LIN {X 0,Y 228.257,Z 260.465,A -85,B 0,C 180,E1 -20025.086,E2 -20025.086} C_VEL
LIN {X 0,Y 228.489,Z 263.113,A -85,B 0,C 180,E1 -20029.335,E2 -20029.335} C_VEL
LIN {X 0,Y 229.645,Z 266.297,A -85,B 0,C 180,E1 -20029.751,E2 -20029.751} C_VEL
LIN {X 0,Y 231.014,Z 268.634,A -85,B 0,C 180,E1 -20030.164,E2 -20030.164} C_VEL
LIN {X 0,Y 235.943,Z 279.475,A -85,B 0,C 180,E1 -20031.89,E2 -20031.89} C_VEL
LIN {X 0,Y 239.913,Z 290.987,A -85,B 0,C 180,E1 -20033.668,E2 -20033.668} C_VEL
LIN {X 0,Y 242.925,Z 302.472,A -85,B 0,C 180,E1 -20035.491,E2 -20035.491} C_VEL
LIN {X 0,Y 244.896,Z 313.256,A -85,B 0,C 180,E1 -20037.287,E2 -20037.287} C_VEL
LIN {X 0,Y 245.991,Z 323.127,A -85,B 0,C 180,E1 -20039.052,E2 -20039.052} C_VEL
LIN {X 0,Y 245.201,Z 327.647,A -85,B 0,C 180,E1 -20039.767,E2 -20039.767} C_VEL
LIN {X 0,Y 242.212,Z 338.615,A -85,B 0,C 180,E1 -20041.632,E2 -20041.632} C_VEL
LIN {X 0,Y 239.048,Z 349.08,A -85,B 0,C 180,E1 -20043.832,E2 -20043.832} C_VEL
LIN {X 0,Y 235.989,Z 358.524,A -85,B 0,C 180,E1 -20046.294,E2 -20046.294} C_VEL
LIN {X 0,Y 233.317,Z 366.346,A -85,B 0,C 180,E1 -20048.81,E2 -20048.81} C_VEL
LIN {X 0,Y 231.34,Z 372.844,A -85,B 0,C 180,E1 -20051.399,E2 -20051.399} C_VEL
LIN {X 0,Y 229.395,Z 378.242,A -85,B 0,C 180,E1 -20053.994,E2 -20053.994} C_VEL
LIN {X 0,Y 227.608,Z 383.911,A -85,B 0,C 180,E1 -20057.518,E2 -20057.518} C_VEL
LIN {X 0,Y 226.471,Z 388.027,A -85,B 0,C 180,E1 -20061.074,E2 -20061.074} C_VEL
LIN {X 0,Y 225.835,Z 390.798,A -85,B 0,C 180,E1 -20064.777,E2 -20064.777} C_VEL
LIN {X 0,Y 225.647,Z 392.058,A -85,B 0,C 180,E1 -20068.215,E2 -20068.215} C_VEL
LIN {X 0,Y 225.667,Z 392.235,A -85,B 0,C 180,E1 -20070,E2 -20070} C_VEL
LIN {X 0,Y 225.703,Z 391.606,A -85,B 0,C 180,E1 -20073.571,E2 -20073.571} C_VEL
LIN {X 0,Y 226.103,Z 389.645,A -85,B 0,C 180,E1 -20077.142,E2 -20077.142} C_VEL
LIN {X 0,Y 226.949,Z 386.307,A -85,B 0,C 180,E1 -20080.708,E2 -20080.708} C_VEL
LIN {X 0,Y 228.318,Z 381.491,A -85,B 0,C 180,E1 -20084.256,E2 -20084.256} C_VEL
LIN {X 0,Y 230.642,Z 375.034,A -85,B 0,C 180,E1 -20087.741,E2 -20087.741} C_VEL
LIN {X 0,Y 232.661,Z 368.29,A -85,B 0,C 180,E1 -20090.606,E2 -20090.606} C_VEL
LIN {X 0,Y 235.407,Z 360.312,A -85,B 0,C 180,E1 -20093.302,E2 -20093.302} C_VEL
LIN {X 0,Y 238.452,Z 351.255,A -85,B 0,C 180,E1 -20095.769,E2 -20095.769} C_VEL
LIN {X 0,Y 241.791,Z 340.283,A -85,B 0,C 180,E1 -20098.186,E2 -20098.186} C_VEL
LIN {X 0,Y 244.745,Z 329.799,A -85,B 0,C 180,E1 -20100.029,E2 -20100.029} C_VEL
LIN {X 0,Y 246.084,Z 323.924,A -85,B 0,C 180,E1 -20100.936,E2 -20100.936} C_VEL
LIN {X 0,Y 245.035,Z 313.632,A -85,B 0,C 180,E1 -20102.773,E2 -20102.773} C_VEL
LIN {X 0,Y 242.991,Z 302.457,A -85,B 0,C 180,E1 -20104.644,E2 -20104.644} C_VEL
LIN {X 0,Y 239.709,Z 289.968,A -85,B 0,C 180,E1 -20106.619,E2 -20106.619} C_VEL
LIN {X 0,Y 235.279,Z 277.883,A -85,B 0,C 180,E1 -20108.509,E2 -20108.509} C_VEL
LIN {X 0,Y 232.127,Z 271.034,A -85,B 0,C 180,E1 -20109.612,E2 -20109.612} C_VEL
LIN {X 0,Y 230.198,Z 267.155,A -85,B 0,C 180,E1 -20110.247,E2 -20110.247} C_VEL
LIN {X 0,Y 228.812,Z 264.447,A -85,B 0,C 180,E1 -20110.674,E2 -20110.674} C_VEL
LIN {X 0,Y 228.503,Z 263.113,A -85,B 0,C 180,E1 -20110.832,E2 -20110.832} C_VEL
LIN {X 0,Y 228.241,Z 260.465,A -85,B 0,C 180,E1 -20115.09,E2 -20115.09} C_VEL
LIN {X 0,Y 227.843,Z 257.899,A -85,B 0,C 180,E1 -20119.627,E2 -20119.627} C_VEL
LIN {X 0,Y 227.867,Z 257.727,A -85,B 0,C 180,E1 -20124.125,E2 -20124.125} C_VEL
LIN {X 0,Y 227.873,Z 257.726,A -85,B 0,C 180,E1 -20128.378,E2 -20128.378} C_VEL
LIN {X 0,Y 227.888,Z 257.724,A -85,B 0,C 180,E1 -20132.445,E2 -20132.445} C_VEL
LIN {X 0,Y 227.909,Z 257.721,A -85,B 0,C 180,E1 -20136.367,E2 -20136.367} C_VEL
LIN {X 0,Y 227.941,Z 257.715,A -85,B 0,C 180,E1 -20140.174,E2 -20140.174} C_VEL
LIN {X 0,Y 228.061,Z 257.701,A -85,B 0,C 180,E1 -20143.898,E2 -20143.898} C_VEL
LIN {X 0,Y 228.075,Z 257.701,A -85,B 0,C 180,E1 -20147.543,E2 -20147.543} C_VEL
LIN {X 0,Y 228.266,Z 257.676,A -85,B 0,C 180,E1 -20151.144,E2 -20151.144} C_VEL
LIN {X 0,Y 228.321,Z 257.67,A -85,B 0,C 180,E1 -20152.927,E2 -20152.927} C_VEL
LIN {X 0,Y 228.552,Z 257.641,A -85,B 0,C 180,E1 -20158.238,E2 -20158.238} C_VEL
LIN {X 0,Y 228.555,Z 257.64,A -85,B 0,C 180,E1 -20161.762,E2 -20161.762} C_VEL
LIN {X 0,Y 228.31,Z 257.669,A -85,B 0,C 180,E1 -20167.073,E2 -20167.073} C_VEL
LIN {X 0,Y 228.145,Z 257.692,A -85,B 0,C 180,E1 -20170.651,E2 -20170.651} C_VEL
LIN {X 0,Y 228.041,Z 257.705,A -85,B 0,C 180,E1 -20174.273,E2 -20174.273} C_VEL
LIN {X 0,Y 227.97,Z 257.715,A -85,B 0,C 180,E1 -20177.956,E2 -20177.956} C_VEL
LIN {X 0,Y 227.922,Z 257.72,A -85,B 0,C 180,E1 -20182.323,E2 -20182.323} C_VEL
LIN {X 0,Y 227.924,Z 257.714,A -85,B 0,C 180,E1 -20186.592,E2 -20186.592} C_VEL
LIN {X 0,Y 227.875,Z 257.726,A -85,B 0,C 180,E1 -20190.28,E2 -20190.28} C_VEL
LIN {X 0,Y 227.857,Z 257.724,A -85,B 0,C 180,E1 -20191.624,E2 -20191.624} C_VEL
LIN {X 0,Y 227.976,Z 258.28,A -85,B 0,C 180,E1 -20193.704,E2 -20193.704} C_VEL
LIN {X 0,Y 228.398,Z 260.942,A -85,B 0,C 180,E1 -20197.982,E2 -20197.982} C_VEL
LIN {X 0,Y 228.903,Z 264.055,A -85,B 0,C 180,E1 -20202.534,E2 -20202.534} C_VEL
LIN {X 0,Y 229.191,Z 265.956,A -85,B 0,C 180,E1 -20205.147,E2 -20205.147} C_VEL
LIN {X 0,Y 229.35,Z 268.73,A -85,B 0,C 180,E1 -20208.665,E2 -20208.665} C_VEL
LIN {X 0,Y 229.788,Z 269.831,A -85,B 0,C 180,E1 -20209.268,E2 -20209.268} C_VEL
LIN {X 0,Y 230.97,Z 272.393,A -85,B 0,C 180,E1 -20209.868,E2 -20209.868} C_VEL
LIN {X 0,Y 232.259,Z 276.618,A -85,B 0,C 180,E1 -20210.386,E2 -20210.386} C_VEL
LIN {X 0,Y 232.855,Z 282.514,A -85,B 0,C 180,E1 -20210.851,E2 -20210.851} C_VEL
LIN {X 0,Y 232.552,Z 288.953,A -85,B 0,C 180,E1 -20211.289,E2 -20211.289} C_VEL
LIN {X 0,Y 232.587,Z 295.048,A -85,B 0,C 180,E1 -20211.896,E2 -20211.896} C_VEL
LIN {X 0,Y 232.958,Z 296.91,A -85,B 0,C 180,E1 -20212.162,E2 -20212.162} C_VEL
LIN {X 0,Y 235.613,Z 308.607,A -85,B 0,C 180,E1 -20213.985,E2 -20213.985} C_VEL
LIN {X 0,Y 237.168,Z 319.32,A -85,B 0,C 180,E1 -20215.734,E2 -20215.734} C_VEL
LIN {X 0,Y 238.014,Z 331.504,A -85,B 0,C 180,E1 -20217.893,E2 -20217.893} C_VEL
LIN {X 0,Y 237.956,Z 336.523,A -85,B 0,C 180,E1 -20218.839,E2 -20218.839} C_VEL
LIN {X 0,Y 234.74,Z 348.029,A -85,B 0,C 180,E1 -20220.888,E2 -20220.888} C_VEL
LIN {X 0,Y 231.105,Z 359.097,A -85,B 0,C 180,E1 -20223.349,E2 -20223.349} C_VEL
LIN {X 0,Y 228.033,Z 368.236,A -85,B 0,C 180,E1 -20225.897,E2 -20225.897} C_VEL
LIN {X 0,Y 225.047,Z 376.976,A -85,B 0,C 180,E1 -20228.953,E2 -20228.953} C_VEL
LIN {X 0,Y 223.05,Z 383.133,A -85,B 0,C 180,E1 -20231.634,E2 -20231.634} C_VEL
LIN {X 0,Y 220.835,Z 389.674,A -85,B 0,C 180,E1 -20235.25,E2 -20235.25} C_VEL
LIN {X 0,Y 219.427,Z 394.573,A -85,B 0,C 180,E1 -20238.92,E2 -20238.92} C_VEL
LIN {X 0,Y 218.684,Z 397.982,A -85,B 0,C 180,E1 -20242.614,E2 -20242.614} C_VEL
LIN {X 0,Y 218.48,Z 399.737,A -85,B 0,C 180,E1 -20245.71,E2 -20245.71} C_VEL
LIN {X 0,Y 218.469,Z 400.5,A -85,B 0,C 180,E1 -20248.156,E2 -20248.156} C_VEL
LIN {X 0,Y 218.574,Z 400.666,A -85,B 0,C 180,E1 -20250,E2 -20250} C_VEL
LIN {X 0,Y 218.449,Z 399.983,A -85,B 0,C 180,E1 -20253.689,E2 -20253.689} C_VEL
LIN {X 0,Y 218.684,Z 397.952,A -85,B 0,C 180,E1 -20257.386,E2 -20257.386} C_VEL
LIN {X 0,Y 219.415,Z 394.525,A -85,B 0,C 180,E1 -20261.08,E2 -20261.08} C_VEL
LIN {X 0,Y 220.828,Z 389.603,A -85,B 0,C 180,E1 -20264.75,E2 -20264.75} C_VEL
LIN {X 0,Y 223.041,Z 383.044,A -85,B 0,C 180,E1 -20268.367,E2 -20268.367} C_VEL
LIN {X 0,Y 225.382,Z 375.745,A -85,B 0,C 180,E1 -20271.493,E2 -20271.493} C_VEL
LIN {X 0,Y 228.498,Z 366.709,A -85,B 0,C 180,E1 -20274.533,E2 -20274.533} C_VEL
LIN {X 0,Y 231.657,Z 357.234,A -85,B 0,C 180,E1 -20277.069,E2 -20277.069} C_VEL
LIN {X 0,Y 235.087,Z 346.749,A -85,B 0,C 180,E1 -20279.31,E2 -20279.31} C_VEL
LIN {X 0,Y 237.729,Z 337.361,A -85,B 0,C 180,E1 -20280.982,E2 -20280.982} C_VEL
LIN {X 0,Y 237.869,Z 329.442,A -85,B 0,C 180,E1 -20282.438,E2 -20282.438} C_VEL
LIN {X 0,Y 236.904,Z 317.539,A -85,B 0,C 180,E1 -20284.513,E2 -20284.513} C_VEL
LIN {X 0,Y 235.241,Z 306.98,A -85,B 0,C 180,E1 -20286.231,E2 -20286.231} C_VEL
LIN {X 0,Y 232.694,Z 296.172,A -85,B 0,C 180,E1 -20287.903,E2 -20287.903} C_VEL
LIN {X 0,Y 229.123,Z 285.061,A -85,B 0,C 180,E1 -20289.607,E2 -20289.607} C_VEL
LIN {X 0,Y 225.78,Z 277.127,A -85,B 0,C 180,E1 -20290.878,E2 -20290.878} C_VEL
LIN {X 0,Y 224.135,Z 273.5,A -85,B 0,C 180,E1 -20291.464,E2 -20291.464} C_VEL
LIN {X 0,Y 222.625,Z 270.595,A -85,B 0,C 180,E1 -20291.953,E2 -20291.953} C_VEL
LIN {X 0,Y 222.315,Z 269.109,A -85,B 0,C 180,E1 -20292.166,E2 -20292.166} C_VEL
LIN {X 0,Y 221.999,Z 266.349,A -85,B 0,C 180,E1 -20295.855,E2 -20295.855} C_VEL
LIN {X 0,Y 221.579,Z 263.09,A -85,B 0,C 180,E1 -20300.628,E2 -20300.628} C_VEL
LIN {X 0,Y 221.102,Z 260.321,A -85,B 0,C 180,E1 -20305.1,E2 -20305.1} C_VEL
LIN {X 0,Y 220.88,Z 259.101,A -85,B 0,C 180,E1 -20307.255,E2 -20307.255} C_VEL
LIN {X 0,Y 220.834,Z 258.604,A -85,B 0,C 180,E1 -20309.39,E2 -20309.39} C_VEL
LIN {X 0,Y 220.876,Z 258.597,A -85,B 0,C 180,E1 -20313.547,E2 -20313.547} C_VEL
LIN {X 0,Y 220.867,Z 258.599,A -85,B 0,C 180,E1 -20317.552,E2 -20317.552} C_VEL
LIN {X 0,Y 220.931,Z 258.586,A -85,B 0,C 180,E1 -20322.617,E2 -20322.617} C_VEL
LIN {X 0,Y 221.004,Z 258.581,A -85,B 0,C 180,E1 -20327.138,E2 -20327.138} C_VEL
LIN {X 0,Y 221.198,Z 258.556,A -85,B 0,C 180,E1 -20330.859,E2 -20330.859} C_VEL
LIN {X 0,Y 221.127,Z 258.565,A -85,B 0,C 180,E1 -20334.529,E2 -20334.529} C_VEL
LIN {X 0,Y 221.511,Z 258.519,A -85,B 0,C 180,E1 -20338.182,E2 -20338.182} C_VEL
LIN {X 0,Y 221.511,Z 258.516,A -85,B 0,C 180,E1 -20341.818,E2 -20341.818} C_VEL
LIN {X 0,Y 221.261,Z 258.549,A -85,B 0,C 180,E1 -20347.3,E2 -20347.3} C_VEL
LIN {X 0,Y 221.083,Z 258.571,A -85,B 0,C 180,E1 -20350.996,E2 -20350.996} C_VEL
LIN {X 0,Y 221.018,Z 258.58,A -85,B 0,C 180,E1 -20356.63,E2 -20356.63} C_VEL
LIN {X 0,Y 220.886,Z 258.594,A -85,B 0,C 180,E1 -20360.487,E2 -20360.487} C_VEL
LIN {X 0,Y 220.864,Z 258.597,A -85,B 0,C 180,E1 -20364.436,E2 -20364.436} C_VEL
LIN {X 0,Y 220.828,Z 258.603,A -85,B 0,C 180,E1 -20368.515,E2 -20368.515} C_VEL
LIN {X 0,Y 220.817,Z 258.604,A -85,B 0,C 180,E1 -20372.756,E2 -20372.756} C_VEL
LIN {X 0,Y 220.802,Z 258.607,A -85,B 0,C 180,E1 -20377.275,E2 -20377.275} C_VEL
LIN {X 0,Y 220.796,Z 258.683,A -85,B 0,C 180,E1 -20379.539,E2 -20379.539} C_VEL
LIN {X 0,Y 221.19,Z 261.272,A -85,B 0,C 180,E1 -20384.349,E2 -20384.349} C_VEL
LIN {X 0,Y 221.465,Z 263.28,A -85,B 0,C 180,E1 -20387.742,E2 -20387.742} C_VEL
LIN {X 0,Y 222.597,Z 266.399,A -85,B 0,C 180,E1 -20388.192,E2 -20388.192} C_VEL
LIN {X 0,Y 224.096,Z 268.756,A -85,B 0,C 180,E1 -20388.667,E2 -20388.667} C_VEL
LIN {X 0,Y 229.315,Z 279.77,A -85,B 0,C 180,E1 -20390.589,E2 -20390.589} C_VEL
LIN {X 0,Y 233.519,Z 291.493,A -85,B 0,C 180,E1 -20392.542,E2 -20392.542} C_VEL
LIN {X 0,Y 236.826,Z 304.525,A -85,B 0,C 180,E1 -20394.721,E2 -20394.721} C_VEL
LIN {X 0,Y 238.737,Z 315.837,A -85,B 0,C 180,E1 -20396.724,E2 -20396.724} C_VEL
LIN {X 0,Y 239.585,Z 325.305,A -85,B 0,C 180,E1 -20398.507,E2 -20398.507} C_VEL
LIN {X 0,Y 236.916,Z 335.554,A -85,B 0,C 180,E1 -20400.206,E2 -20400.206} C_VEL
LIN {X 0,Y 233.85,Z 345.666,A -85,B 0,C 180,E1 -20402.236,E2 -20402.236} C_VEL
LIN {X 0,Y 230.562,Z 355.7,A -85,B 0,C 180,E1 -20404.739,E2 -20404.739} C_VEL
LIN {X 0,Y 227.557,Z 364.031,A -85,B 0,C 180,E1 -20407.291,E2 -20407.291} C_VEL
LIN {X 0,Y 224.829,Z 371.981,A -85,B 0,C 180,E1 -20410.364,E2 -20410.364} C_VEL
LIN {X 0,Y 223.217,Z 376.707,A -85,B 0,C 180,E1 -20412.596,E2 -20412.596} C_VEL
LIN {X 0,Y 221.447,Z 381.418,A -85,B 0,C 180,E1 -20415.292,E2 -20415.292} C_VEL
LIN {X 0,Y 219.965,Z 386.291,A -85,B 0,C 180,E1 -20418.948,E2 -20418.948} C_VEL
LIN {X 0,Y 219.049,Z 389.679,A -85,B 0,C 180,E1 -20422.627,E2 -20422.627} C_VEL
LIN {X 0,Y 218.622,Z 391.687,A -85,B 0,C 180,E1 -20426.314,E2 -20426.314} C_VEL
LIN {X 0,Y 218.585,Z 392.369,A -85,B 0,C 180,E1 -20430,E2 -20430} C_VEL
LIN {X 0,Y 218.62,Z 391.74,A -85,B 0,C 180,E1 -20433.687,E2 -20433.687} C_VEL
LIN {X 0,Y 219.049,Z 389.78,A -85,B 0,C 180,E1 -20437.374,E2 -20437.374} C_VEL
LIN {X 0,Y 219.951,Z 386.442,A -85,B 0,C 180,E1 -20441.053,E2 -20441.053} C_VEL
LIN {X 0,Y 221.41,Z 381.625,A -85,B 0,C 180,E1 -20444.711,E2 -20444.711} C_VEL
LIN {X 0,Y 223.874,Z 375.168,A -85,B 0,C 180,E1 -20448.296,E2 -20448.296} C_VEL
LIN {X 0,Y 225.91,Z 368.651,A -85,B 0,C 180,E1 -20451.154,E2 -20451.154} C_VEL
LIN {X 0,Y 228.901,Z 360.444,A -85,B 0,C 180,E1 -20454.005,E2 -20454.005} C_VEL
LIN {X 0,Y 232.053,Z 351.388,A -85,B 0,C 180,E1 -20456.534,E2 -20456.534} C_VEL
LIN {X 0,Y 235.555,Z 340.414,A -85,B 0,C 180,E1 -20459.002,E2 -20459.002} C_VEL
LIN {X 0,Y 238.814,Z 329.133,A -85,B 0,C 180,E1 -20461.014,E2 -20461.014} C_VEL
LIN {X 0,Y 239.666,Z 324.668,A -85,B 0,C 180,E1 -20461.744,E2 -20461.744} C_VEL
LIN {X 0,Y 238.534,Z 313.568,A -85,B 0,C 180,E1 -20463.818,E2 -20463.818} C_VEL
LIN {X 0,Y 236.426,Z 302.352,A -85,B 0,C 180,E1 -20465.784,E2 -20465.784} C_VEL
LIN {X 0,Y 233.712,Z 292.001,A -85,B 0,C 180,E1 -20467.52,E2 -20467.52} C_VEL
LIN {X 0,Y 229.307,Z 279.636,A -85,B 0,C 180,E1 -20469.58,E2 -20469.58} C_VEL
LIN {X 0,Y 225.292,Z 271.3,A -85,B 0,C 180,E1 -20471.058,E2 -20471.058} C_VEL
LIN {X 0,Y 223.483,Z 267.64,A -85,B 0,C 180,E1 -20471.703,E2 -20471.703} C_VEL
LIN {X 0,Y 221.854,Z 264.855,A -85,B 0,C 180,E1 -20472.224,E2 -20472.224} C_VEL
LIN {X 0,Y 221.446,Z 263.285,A -85,B 0,C 180,E1 -20472.425,E2 -20472.425} C_VEL
LIN {X 0,Y 221.076,Z 260.645,A -85,B 0,C 180,E1 -20476.985,E2 -20476.985} C_VEL
LIN {X 0,Y 220.812,Z 258.778,A -85,B 0,C 180,E1 -20480.464,E2 -20480.464} C_VEL
LIN {X 0,Y 220.826,Z 258.604,A -85,B 0,C 180,E1 -20482.793,E2 -20482.793} C_VEL
LIN {X 0,Y 220.82,Z 258.605,A -85,B 0,C 180,E1 -20487.244,E2 -20487.244} C_VEL
LIN {X 0,Y 220.839,Z 258.602,A -85,B 0,C 180,E1 -20491.487,E2 -20491.487} C_VEL
LIN {X 0,Y 220.865,Z 258.593,A -85,B 0,C 180,E1 -20495.565,E2 -20495.565} C_VEL
LIN {X 0,Y 220.888,Z 258.594,A -85,B 0,C 180,E1 -20499.513,E2 -20499.513} C_VEL
LIN {X 0,Y 221.019,Z 258.58,A -85,B 0,C 180,E1 -20503.37,E2 -20503.37} C_VEL
LIN {X 0,Y 221.014,Z 258.578,A -85,B 0,C 180,E1 -20507.139,E2 -20507.139} C_VEL
LIN {X 0,Y 221.204,Z 258.556,A -85,B 0,C 180,E1 -20510.859,E2 -20510.859} C_VEL
LIN {X 0,Y 221.257,Z 258.549,A -85,B 0,C 180,E1 -20512.7,E2 -20512.7} C_VEL
LIN {X 0,Y 221.51,Z 258.518,A -85,B 0,C 180,E1 -20518.182,E2 -20518.182} C_VEL
LIN {X 0,Y 221.513,Z 258.517,A -85,B 0,C 180,E1 -20521.818,E2 -20521.818} C_VEL
LIN {X 0,Y 221.247,Z 258.549,A -85,B 0,C 180,E1 -20527.3,E2 -20527.3} C_VEL
LIN {X 0,Y 221.065,Z 258.575,A -85,B 0,C 180,E1 -20530.996,E2 -20530.996} C_VEL
LIN {X 0,Y 220.988,Z 258.582,A -85,B 0,C 180,E1 -20536.632,E2 -20536.632} C_VEL
LIN {X 0,Y 220.882,Z 258.596,A -85,B 0,C 180,E1 -20540.487,E2 -20540.487} C_VEL
LIN {X 0,Y 220.849,Z 258.598,A -85,B 0,C 180,E1 -20544.437,E2 -20544.437} C_VEL
LIN {X 0,Y 220.806,Z 258.605,A -85,B 0,C 180,E1 -20548.518,E2 -20548.518} C_VEL
LIN {X 0,Y 220.82,Z 258.602,A -85,B 0,C 180,E1 -20550.758,E2 -20550.758} C_VEL
LIN {X 0,Y 220.894,Z 259.155,A -85,B 0,C 180,E1 -20552.743,E2 -20552.743} C_VEL
LIN {X 0,Y 221.399,Z 261.939,A -85,B 0,C 180,E1 -20557.477,E2 -20557.477} C_VEL
LIN {X 0,Y 221.797,Z 264.734,A -85,B 0,C 180,E1 -20561.714,E2 -20561.714} C_VEL
LIN {X 0,Y 222.221,Z 267.707,A -85,B 0,C 180,E1 -20565.911,E2 -20565.911} C_VEL
LIN {X 0,Y 222.335,Z 269.174,A -85,B 0,C 180,E1 -20567.836,E2 -20567.836} C_VEL
LIN {X 0,Y 223.344,Z 272.251,A -85,B 0,C 180,E1 -20568.223,E2 -20568.223} C_VEL
LIN {X 0,Y 224.813,Z 274.705,A -85,B 0,C 180,E1 -20568.683,E2 -20568.683} C_VEL
LIN {X 0,Y 229.334,Z 285.417,A -85,B 0,C 180,E1 -20570.399,E2 -20570.399} C_VEL
LIN {X 0,Y 232.958,Z 296.91,A -85,B 0,C 180,E1 -20572.162,E2 -20572.162} C_VEL
LIN {X 0,Y 233.805,Z 302.011,A -85,B 0,C 180,E1 -20572.867,E2 -20572.867} C_VEL
LIN {X 0,Y 233.669,Z 307.392,A -85,B 0,C 180,E1 -20573.483,E2 -20573.483} C_VEL
LIN {X 0,Y 231.828,Z 318.322,A -85,B 0,C 180,E1 -20574.699,E2 -20574.699} C_VEL
LIN {X 0,Y 231.236,Z 323.452,A -85,B 0,C 180,E1 -20575.428,E2 -20575.428} C_VEL
LIN {X 0,Y 231.257,Z 325.088,A -85,B 0,C 180,E1 -20575.704,E2 -20575.704} C_VEL
LIN {X 0,Y 231.615,Z 336.926,A -85,B 0,C 180,E1 -20577.992,E2 -20577.992} C_VEL
LIN {X 0,Y 228.544,Z 347.897,A -85,B 0,C 180,E1 -20580.019,E2 -20580.019} C_VEL
LIN {X 0,Y 224.74,Z 358.964,A -85,B 0,C 180,E1 -20582.531,E2 -20582.531} C_VEL
LIN {X 0,Y 221.544,Z 368.103,A -85,B 0,C 180,E1 -20585.144,E2 -20585.144} C_VEL
LIN {X 0,Y 218.375,Z 376.841,A -85,B 0,C 180,E1 -20588.278,E2 -20588.278} C_VEL
LIN {X 0,Y 216.272,Z 382.999,A -85,B 0,C 180,E1 -20591.037,E2 -20591.037} C_VEL
LIN {X 0,Y 213.926,Z 389.539,A -85,B 0,C 180,E1 -20594.762,E2 -20594.762} C_VEL
LIN {X 0,Y 212.413,Z 394.438,A -85,B 0,C 180,E1 -20598.549,E2 -20598.549} C_VEL
LIN {X 0,Y 211.624,Z 397.848,A -85,B 0,C 180,E1 -20602.366,E2 -20602.366} C_VEL
LIN {X 0,Y 211.387,Z 399.734,A -85,B 0,C 180,E1 -20605.876,E2 -20605.876} C_VEL
LIN {X 0,Y 211.373,Z 400.366,A -85,B 0,C 180,E1 -20608.094,E2 -20608.094} C_VEL
LIN {X 0,Y 211.473,Z 400.531,A -85,B 0,C 180,E1 -20610,E2 -20610} C_VEL
LIN {X 0,Y 211.355,Z 399.848,A -85,B 0,C 180,E1 -20613.813,E2 -20613.813} C_VEL
LIN {X 0,Y 211.623,Z 397.816,A -85,B 0,C 180,E1 -20617.634,E2 -20617.634} C_VEL
LIN {X 0,Y 212.403,Z 394.389,A -85,B 0,C 180,E1 -20621.451,E2 -20621.451} C_VEL
LIN {X 0,Y 213.918,Z 389.466,A -85,B 0,C 180,E1 -20625.238,E2 -20625.238} C_VEL
LIN {X 0,Y 216.25,Z 382.906,A -85,B 0,C 180,E1 -20628.965,E2 -20628.965} C_VEL
LIN {X 0,Y 218.744,Z 375.607,A -85,B 0,C 180,E1 -20632.18,E2 -20632.18} C_VEL
LIN {X 0,Y 222.02,Z 366.571,A -85,B 0,C 180,E1 -20635.299,E2 -20635.299} C_VEL
LIN {X 0,Y 225.351,Z 357.096,A -85,B 0,C 180,E1 -20637.892,E2 -20637.892} C_VEL
LIN {X 0,Y 228.902,Z 346.61,A -85,B 0,C 180,E1 -20640.183,E2 -20640.183} C_VEL
LIN {X 0,Y 231.49,Z 337.213,A -85,B 0,C 180,E1 -20641.915,E2 -20641.915} C_VEL
LIN {X 0,Y 231.394,Z 328.133,A -85,B 0,C 180,E1 -20643.673,E2 -20643.673} C_VEL
LIN {X 0,Y 230.364,Z 315.879,A -85,B 0,C 180,E1 -20645.866,E2 -20645.866} C_VEL
LIN {X 0,Y 227.971,Z 302.859,A -85,B 0,C 180,E1 -20648.066,E2 -20648.066} C_VEL
LIN {X 0,Y 224.423,Z 290.267,A -85,B 0,C 180,E1 -20650.138,E2 -20650.138} C_VEL
LIN {X 0,Y 221.139,Z 281.733,A -85,B 0,C 180,E1 -20651.597,E2 -20651.597} C_VEL
LIN {X 0,Y 219.109,Z 277.353,A -85,B 0,C 180,E1 -20652.377,E2 -20652.377} C_VEL
LIN {X 0,Y 217.402,Z 273.701,A -85,B 0,C 180,E1 -20653.031,E2 -20653.031} C_VEL
LIN {X 0,Y 215.582,Z 270.586,A -85,B 0,C 180,E1 -20653.648,E2 -20653.648} C_VEL
LIN {X 0,Y 215.179,Z 268.976,A -85,B 0,C 180,E1 -20653.839,E2 -20653.839} C_VEL
LIN {X 0,Y 214.947,Z 266.999,A -85,B 0,C 180,E1 -20656.636,E2 -20656.636} C_VEL
LIN {X 0,Y 214.497,Z 263.841,A -85,B 0,C 180,E1 -20661.499,E2 -20661.499} C_VEL
LIN {X 0,Y 214.049,Z 261.162,A -85,B 0,C 180,E1 -20666.071,E2 -20666.071} C_VEL
LIN {X 0,Y 213.781,Z 259.741,A -85,B 0,C 180,E1 -20668.731,E2 -20668.731} C_VEL
LIN {X 0,Y 213.789,Z 259.481,A -85,B 0,C 180,E1 -20672.598,E2 -20672.598} C_VEL
LIN {X 0,Y 213.811,Z 259.478,A -85,B 0,C 180,E1 -20676.979,E2 -20676.979} C_VEL
LIN {X 0,Y 213.888,Z 259.463,A -85,B 0,C 180,E1 -20682.344,E2 -20682.344} C_VEL
LIN {X 0,Y 213.943,Z 259.458,A -85,B 0,C 180,E1 -20686.706,E2 -20686.706} C_VEL
LIN {X 0,Y 214.137,Z 259.432,A -85,B 0,C 180,E1 -20690.555,E2 -20690.555} C_VEL
LIN {X 0,Y 214.089,Z 259.442,A -85,B 0,C 180,E1 -20694.348,E2 -20694.348} C_VEL
LIN {X 0,Y 214.444,Z 259.399,A -85,B 0,C 180,E1 -20698.122,E2 -20698.122} C_VEL
LIN {X 0,Y 214.54,Z 259.386,A -85,B 0,C 180,E1 -20700,E2 -20700} C_VEL
LIN {X 0,Y 214.444,Z 259.397,A -85,B 0,C 180,E1 -20701.878,E2 -20701.878} C_VEL
LIN {X 0,Y 214.2,Z 259.428,A -85,B 0,C 180,E1 -20707.542,E2 -20707.542} C_VEL
LIN {X 0,Y 214.009,Z 259.451,A -85,B 0,C 180,E1 -20711.364,E2 -20711.364} C_VEL
LIN {X 0,Y 213.936,Z 259.462,A -85,B 0,C 180,E1 -20715.237,E2 -20715.237} C_VEL
LIN {X 0,Y 213.838,Z 259.475,A -85,B 0,C 180,E1 -20719.188,E2 -20719.188} C_VEL
LIN {X 0,Y 213.812,Z 259.477,A -85,B 0,C 180,E1 -20723.231,E2 -20723.231} C_VEL
LIN {X 0,Y 213.83,Z 259.473,A -85,B 0,C 180,E1 -20727.45,E2 -20727.45} C_VEL
LIN {X 0,Y 213.768,Z 259.482,A -85,B 0,C 180,E1 -20731.738,E2 -20731.738} C_VEL
LIN {X 0,Y 213.742,Z 259.487,A -85,B 0,C 180,E1 -20736.289,E2 -20736.289} C_VEL
LIN {X 0,Y 213.739,Z 259.59,A -85,B 0,C 180,E1 -20738.664,E2 -20738.664} C_VEL
LIN {X 0,Y 214.125,Z 262.118,A -85,B 0,C 180,E1 -20743.572,E2 -20743.572} C_VEL
LIN {X 0,Y 214.311,Z 263.487,A -85,B 0,C 180,E1 -20746.007,E2 -20746.007} C_VEL
LIN {X 0,Y 215.331,Z 266.331,A -85,B 0,C 180,E1 -20746.423,E2 -20746.423} C_VEL
LIN {X 0,Y 217.222,Z 269.087,A -85,B 0,C 180,E1 -20747.061,E2 -20747.061} C_VEL
LIN {X 0,Y 221.851,Z 278.418,A -85,B 0,C 180,E1 -20748.857,E2 -20748.857} C_VEL
LIN {X 0,Y 225.509,Z 287.223,A -85,B 0,C 180,E1 -20750.474,E2 -20750.474} C_VEL
LIN {X 0,Y 228.61,Z 297.331,A -85,B 0,C 180,E1 -20752.266,E2 -20752.266} C_VEL
LIN {X 0,Y 231.44,Z 310.225,A -85,B 0,C 180,E1 -20754.593,E2 -20754.593} C_VEL
LIN {X 0,Y 232.882,Z 321.626,A -85,B 0,C 180,E1 -20756.769,E2 -20756.769} C_VEL
LIN {X 0,Y 233.11,Z 327.42,A -85,B 0,C 180,E1 -20757.919,E2 -20757.919} C_VEL
LIN {X 0,Y 229.788,Z 338.892,A -85,B 0,C 180,E1 -20759.946,E2 -20759.946} C_VEL
LIN {X 0,Y 226.374,Z 349.356,A -85,B 0,C 180,E1 -20762.245,E2 -20762.245} C_VEL
LIN {X 0,Y 223.029,Z 358.799,A -85,B 0,C 180,E1 -20764.824,E2 -20764.824} C_VEL
LIN {X 0,Y 219.628,Z 367.845,A -85,B 0,C 180,E1 -20767.934,E2 -20767.934} C_VEL
LIN {X 0,Y 217.172,Z 375.043,A -85,B 0,C 180,E1 -20771.118,E2 -20771.118} C_VEL
LIN {X 0,Y 214.559,Z 381.555,A -85,B 0,C 180,E1 -20774.809,E2 -20774.809} C_VEL
LIN {X 0,Y 212.986,Z 386.427,A -85,B 0,C 180,E1 -20778.581,E2 -20778.581} C_VEL
LIN {X 0,Y 211.995,Z 389.814,A -85,B 0,C 180,E1 -20782.38,E2 -20782.38} C_VEL
LIN {X 0,Y 211.545,Z 391.822,A -85,B 0,C 180,E1 -20786.19,E2 -20786.19} C_VEL
LIN {X 0,Y 211.485,Z 392.504,A -85,B 0,C 180,E1 -20790,E2 -20790} C_VEL
LIN {X 0,Y 211.545,Z 391.874,A -85,B 0,C 180,E1 -20793.81,E2 -20793.81} C_VEL
LIN {X 0,Y 211.995,Z 389.914,A -85,B 0,C 180,E1 -20797.62,E2 -20797.62} C_VEL
LIN {X 0,Y 212.97,Z 386.576,A -85,B 0,C 180,E1 -20801.42,E2 -20801.42} C_VEL
LIN {X 0,Y 214.518,Z 381.76,A -85,B 0,C 180,E1 -20805.195,E2 -20805.195} C_VEL
LIN {X 0,Y 217.12,Z 375.302,A -85,B 0,C 180,E1 -20808.887,E2 -20808.887} C_VEL
LIN {X 0,Y 219.101,Z 369.24,A -85,B 0,C 180,E1 -20811.642,E2 -20811.642} C_VEL
LIN {X 0,Y 222.415,Z 360.577,A -85,B 0,C 180,E1 -20814.752,E2 -20814.752} C_VEL
LIN {X 0,Y 225.707,Z 351.52,A -85,B 0,C 180,E1 -20817.341,E2 -20817.341} C_VEL
LIN {X 0,Y 228.685,Z 342.497,A -85,B 0,C 180,E1 -20819.454,E2 -20819.454} C_VEL
LIN {X 0,Y 232.269,Z 331.06,A -85,B 0,C 180,E1 -20821.607,E2 -20821.607} C_VEL
LIN {X 0,Y 233.124,Z 327.889,A -85,B 0,C 180,E1 -20822.13,E2 -20822.13} C_VEL
LIN {X 0,Y 233.194,Z 324.202,A -85,B 0,C 180,E1 -20822.853,E2 -20822.853} C_VEL
LIN {X 0,Y 231.908,Z 312.301,A -85,B 0,C 180,E1 -20825.156,E2 -20825.156} C_VEL
LIN {X 0,Y 229.229,Z 299.464,A -85,B 0,C 180,E1 -20827.504,E2 -20827.504} C_VEL
LIN {X 0,Y 225.387,Z 286.755,A -85,B 0,C 180,E1 -20829.756,E2 -20829.756} C_VEL
LIN {X 0,Y 221.037,Z 276.494,A -85,B 0,C 180,E1 -20831.653,E2 -20831.653} C_VEL
LIN {X 0,Y 218.499,Z 271.705,A -85,B 0,C 180,E1 -20832.612,E2 -20832.612} C_VEL
LIN {X 0,Y 216.63,Z 268.103,A -85,B 0,C 180,E1 -20833.321,E2 -20833.321} C_VEL
LIN {X 0,Y 214.771,Z 265.197,A -85,B 0,C 180,E1 -20833.952,E2 -20833.952} C_VEL
LIN {X 0,Y 214.297,Z 263.434,A -85,B 0,C 180,E1 -20834.24,E2 -20834.24} C_VEL
LIN {X 0,Y 213.919,Z 260.814,A -85,B 0,C 180,E1 -20839.081,E2 -20839.081} C_VEL
LIN {X 0,Y 213.722,Z 259.489,A -85,B 0,C 180,E1 -20842.113,E2 -20842.113} C_VEL
LIN {X 0,Y 213.757,Z 259.485,A -85,B 0,C 180,E1 -20846.018,E2 -20846.018} C_VEL
LIN {X 0,Y 213.783,Z 259.481,A -85,B 0,C 180,E1 -20850.454,E2 -20850.454} C_VEL
LIN {X 0,Y 213.801,Z 259.471,A -85,B 0,C 180,E1 -20854.701,E2 -20854.701} C_VEL
LIN {X 0,Y 213.807,Z 259.479,A -85,B 0,C 180,E1 -20858.803,E2 -20858.803} C_VEL
LIN {X 0,Y 213.947,Z 259.461,A -85,B 0,C 180,E1 -20862.804,E2 -20862.804} C_VEL
LIN {X 0,Y 213.956,Z 259.457,A -85,B 0,C 180,E1 -20866.707,E2 -20866.707} C_VEL
LIN {X 0,Y 214.142,Z 259.437,A -85,B 0,C 180,E1 -20870.555,E2 -20870.555} C_VEL
LIN {X 0,Y 214.097,Z 259.439,A -85,B 0,C 180,E1 -20874.348,E2 -20874.348} C_VEL
LIN {X 0,Y 214.444,Z 259.398,A -85,B 0,C 180,E1 -20878.122,E2 -20878.122} C_VEL
LIN {X 0,Y 214.446,Z 259.396,A -85,B 0,C 180,E1 -20881.878,E2 -20881.878} C_VEL
LIN {X 0,Y 214.188,Z 259.428,A -85,B 0,C 180,E1 -20887.542,E2 -20887.542} C_VEL
LIN {X 0,Y 213.996,Z 259.456,A -85,B 0,C 180,E1 -20891.364,E2 -20891.364} C_VEL
LIN {X 0,Y 213.908,Z 259.467,A -85,B 0,C 180,E1 -20895.239,E2 -20895.239} C_VEL
LIN {X 0,Y 213.822,Z 259.475,A -85,B 0,C 180,E1 -20899.189,E2 -20899.189} C_VEL
LIN {X 0,Y 213.804,Z 259.477,A -85,B 0,C 180,E1 -20903.232,E2 -20903.232} C_VEL
LIN {X 0,Y 213.789,Z 259.48,A -85,B 0,C 180,E1 -20907.428,E2 -20907.428} C_VEL
LIN {X 0,Y 213.814,Z 259.8,A -85,B 0,C 180,E1 -20911.282,E2 -20911.282} C_VEL
LIN {X 0,Y 214.177,Z 261.741,A -85,B 0,C 180,E1 -20914.88,E2 -20914.88} C_VEL
LIN {X 0,Y 214.508,Z 263.894,A -85,B 0,C 180,E1 -20918.499,E2 -20918.499} C_VEL
LIN {X 0,Y 214.974,Z 267.077,A -85,B 0,C 180,E1 -20923.357,E2 -20923.357} C_VEL
LIN {X 0,Y 215.24,Z 268.987,A -85,B 0,C 180,E1 -20926.075,E2 -20926.075} C_VEL
LIN {X 0,Y 216.477,Z 272.364,A -85,B 0,C 180,E1 -20926.593,E2 -20926.593} C_VEL
LIN {X 0,Y 217.94,Z 274.692,A -85,B 0,C 180,E1 -20927.085,E2 -20927.085} C_VEL
LIN {X 0,Y 222.098,Z 283.868,A -85,B 0,C 180,E1 -20928.723,E2 -20928.723} C_VEL
LIN {X 0,Y 225.591,Z 293.743,A -85,B 0,C 180,E1 -20930.371,E2 -20930.371} C_VEL
LIN {X 0,Y 228.626,Z 305.586,A -85,B 0,C 180,E1 -20932.331,E2 -20932.331} C_VEL
LIN {X 0,Y 230.604,Z 317.511,A -85,B 0,C 180,E1 -20934.365,E2 -20934.365} C_VEL
LIN {X 0,Y 231.257,Z 325.088,A -85,B 0,C 180,E1 -20935.704,E2 -20935.704} C_VEL
LIN {X 0,Y 231.074,Z 328.369,A -85,B 0,C 180,E1 -20936.242,E2 -20936.242} C_VEL
LIN {X 0,Y 230.278,Z 331.692,A -85,B 0,C 180,E1 -20936.734,E2 -20936.734} C_VEL
LIN {X 0,Y 227.514,Z 338.235,A -85,B 0,C 180,E1 -20937.643,E2 -20937.643} C_VEL
LIN {X 0,Y 222.577,Z 347.801,A -85,B 0,C 180,E1 -20939.137,E2 -20939.137} C_VEL
LIN {X 0,Y 221.351,Z 350.783,A -85,B 0,C 180,E1 -20939.752,E2 -20939.752} C_VEL
LIN {X 0,Y 217.85,Z 360.463,A -85,B 0,C 180,E1 -20942.109,E2 -20942.109} C_VEL
LIN {X 0,Y 214.562,Z 369.328,A -85,B 0,C 180,E1 -20944.797,E2 -20944.797} C_VEL
LIN {X 0,Y 211.339,Z 377.828,A -85,B 0,C 180,E1 -20948.03,E2 -20948.03} C_VEL
LIN {X 0,Y 208.822,Z 384.682,A -85,B 0,C 180,E1 -20951.353,E2 -20951.353} C_VEL
LIN {X 0,Y 207.04,Z 389.405,A -85,B 0,C 180,E1 -20954.243,E2 -20954.243} C_VEL
LIN {X 0,Y 205.422,Z 394.304,A -85,B 0,C 180,E1 -20958.154,E2 -20958.154} C_VEL
LIN {X 0,Y 204.56,Z 397.713,A -85,B 0,C 180,E1 -20962.101,E2 -20962.101} C_VEL
LIN {X 0,Y 204.267,Z 399.73,A -85,B 0,C 180,E1 -20966.054,E2 -20966.054} C_VEL
LIN {X 0,Y 204.374,Z 400.397,A -85,B 0,C 180,E1 -20970,E2 -20970} C_VEL
LIN {X 0,Y 204.266,Z 399.713,A -85,B 0,C 180,E1 -20973.946,E2 -20973.946} C_VEL
LIN {X 0,Y 204.559,Z 397.68,A -85,B 0,C 180,E1 -20977.899,E2 -20977.899} C_VEL
LIN {X 0,Y 205.413,Z 394.252,A -85,B 0,C 180,E1 -20981.846,E2 -20981.846} C_VEL
LIN {X 0,Y 207.033,Z 389.33,A -85,B 0,C 180,E1 -20985.758,E2 -20985.758} C_VEL
LIN {X 0,Y 209.464,Z 382.769,A -85,B 0,C 180,E1 -20989.604,E2 -20989.604} C_VEL
LIN {X 0,Y 212.141,Z 375.47,A -85,B 0,C 180,E1 -20992.909,E2 -20992.909} C_VEL
LIN {X 0,Y 215.6,Z 366.434,A -85,B 0,C 180,E1 -20996.108,E2 -20996.108} C_VEL
LIN {X 0,Y 219.068,Z 356.958,A -85,B 0,C 180,E1 -20998.765,E2 -20998.765} C_VEL
LIN {X 0,Y 222.77,Z 346.472,A -85,B 0,C 180,E1 -21001.105,E2 -21001.105} C_VEL
LIN {X 0,Y 225.011,Z 339.035,A -85,B 0,C 180,E1 -21002.508,E2 -21002.508} C_VEL
LIN {X 0,Y 225.105,Z 329.76,A -85,B 0,C 180,E1 -21004.411,E2 -21004.411} C_VEL
LIN {X 0,Y 224.367,Z 318.642,A -85,B 0,C 180,E1 -21006.523,E2 -21006.523} C_VEL
LIN {X 0,Y 222.39,Z 306.363,A -85,B 0,C 180,E1 -21008.734,E2 -21008.734} C_VEL
LIN {X 0,Y 219.368,Z 294.588,A -85,B 0,C 180,E1 -21010.81,E2 -21010.81} C_VEL
LIN {X 0,Y 216.073,Z 285.461,A -85,B 0,C 180,E1 -21012.468,E2 -21012.468} C_VEL
LIN {X 0,Y 212.525,Z 277.83,A -85,B 0,C 180,E1 -21013.97,E2 -21013.97} C_VEL
LIN {X 0,Y 210.51,Z 273.807,A -85,B 0,C 180,E1 -21014.789,E2 -21014.789} C_VEL
LIN {X 0,Y 208.641,Z 270.905,A -85,B 0,C 180,E1 -21015.464,E2 -21015.464} C_VEL
LIN {X 0,Y 208.011,Z 268.798,A -85,B 0,C 180,E1 -21015.763,E2 -21015.763} C_VEL
LIN {X 0,Y 207.602,Z 266.092,A -85,B 0,C 180,E1 -21019.968,E2 -21019.968} C_VEL
LIN {X 0,Y 207.231,Z 263.425,A -85,B 0,C 180,E1 -21024.482,E2 -21024.482} C_VEL
LIN {X 0,Y 206.763,Z 260.877,A -85,B 0,C 180,E1 -21029.346,E2 -21029.346} C_VEL
LIN {X 0,Y 206.71,Z 260.362,A -85,B 0,C 180,E1 -21032.127,E2 -21032.127} C_VEL
LIN {X 0,Y 206.746,Z 260.359,A -85,B 0,C 180,E1 -21036.61,E2 -21036.61} C_VEL
LIN {X 0,Y 206.827,Z 260.342,A -85,B 0,C 180,E1 -21042.193,E2 -21042.193} C_VEL
LIN {X 0,Y 206.883,Z 260.335,A -85,B 0,C 180,E1 -21046.244,E2 -21046.244} C_VEL
LIN {X 0,Y 207.081,Z 260.309,A -85,B 0,C 180,E1 -21050.23,E2 -21050.23} C_VEL
LIN {X 0,Y 207.051,Z 260.319,A -85,B 0,C 180,E1 -21054.156,E2 -21054.156} C_VEL
LIN {X 0,Y 207.381,Z 260.279,A -85,B 0,C 180,E1 -21058.058,E2 -21058.058} C_VEL
LIN {X 0,Y 207.506,Z 260.262,A -85,B 0,C 180,E1 -21060,E2 -21060} C_VEL
LIN {X 0,Y 207.38,Z 260.276,A -85,B 0,C 180,E1 -21061.942,E2 -21061.942} C_VEL
LIN {X 0,Y 207.142,Z 260.308,A -85,B 0,C 180,E1 -21067.8,E2 -21067.8} C_VEL
LIN {X 0,Y 206.933,Z 260.333,A -85,B 0,C 180,E1 -21071.758,E2 -21071.758} C_VEL
LIN {X 0,Y 206.869,Z 260.341,A -85,B 0,C 180,E1 -21075.771,E2 -21075.771} C_VEL
LIN {X 0,Y 206.765,Z 260.353,A -85,B 0,C 180,E1 -21079.871,E2 -21079.871} C_VEL
LIN {X 0,Y 206.748,Z 260.355,A -85,B 0,C 180,E1 -21084.074,E2 -21084.074} C_VEL
LIN {X 0,Y 206.738,Z 260.358,A -85,B 0,C 180,E1 -21088.42,E2 -21088.42} C_VEL
LIN {X 0,Y 206.699,Z 260.362,A -85,B 0,C 180,E1 -21092.958,E2 -21092.958} C_VEL
LIN {X 0,Y 206.7,Z 260.363,A -85,B 0,C 180,E1 -21095.311,E2 -21095.311} C_VEL
LIN {X 0,Y 206.69,Z 260.519,A -85,B 0,C 180,E1 -21097.738,E2 -21097.738} C_VEL
LIN {X 0,Y 207.041,Z 262.966,A -85,B 0,C 180,E1 -21102.758,E2 -21102.758} C_VEL
LIN {X 0,Y 207.207,Z 263.679,A -85,B 0,C 180,E1 -21104.077,E2 -21104.077} C_VEL
LIN {X 0,Y 208.279,Z 266.575,A -85,B 0,C 180,E1 -21104.549,E2 -21104.549} C_VEL
LIN {X 0,Y 210.329,Z 269.535,A -85,B 0,C 180,E1 -21105.307,E2 -21105.307} C_VEL
LIN {X 0,Y 212.346,Z 273.081,A -85,B 0,C 180,E1 -21106.105,E2 -21106.105} C_VEL
LIN {X 0,Y 216.803,Z 282.196,A -85,B 0,C 180,E1 -21108.008,E2 -21108.008} C_VEL
LIN {X 0,Y 220.481,Z 291.922,A -85,B 0,C 180,E1 -21109.909,E2 -21109.909} C_VEL
LIN {X 0,Y 223.375,Z 302.264,A -85,B 0,C 180,E1 -21111.866,E2 -21111.866} C_VEL
LIN {X 0,Y 225.609,Z 313.764,A -85,B 0,C 180,E1 -21114.09,E2 -21114.09} C_VEL
LIN {X 0,Y 226.628,Z 323.578,A -85,B 0,C 180,E1 -21116.069,E2 -21116.069} C_VEL
LIN {X 0,Y 226.838,Z 328.307,A -85,B 0,C 180,E1 -21117.074,E2 -21117.074} C_VEL
LIN {X 0,Y 223.344,Z 340.096,A -85,B 0,C 180,E1 -21119.247,E2 -21119.247} C_VEL
LIN {X 0,Y 220.113,Z 349.494,A -85,B 0,C 180,E1 -21121.384,E2 -21121.384} C_VEL
LIN {X 0,Y 216.612,Z 358.936,A -85,B 0,C 180,E1 -21124.023,E2 -21124.023} C_VEL
LIN {X 0,Y 213.519,Z 366.758,A -85,B 0,C 180,E1 -21126.735,E2 -21126.735} C_VEL
LIN {X 0,Y 211.074,Z 373.257,A -85,B 0,C 180,E1 -21129.536,E2 -21129.536} C_VEL
LIN {X 0,Y 208.967,Z 378.651,A -85,B 0,C 180,E1 -21132.381,E2 -21132.381} C_VEL
LIN {X 0,Y 207.221,Z 383.086,A -85,B 0,C 180,E1 -21135.264,E2 -21135.264} C_VEL
LIN {X 0,Y 206.022,Z 386.563,A -85,B 0,C 180,E1 -21138.19,E2 -21138.19} C_VEL
LIN {X 0,Y 204.937,Z 389.95,A -85,B 0,C 180,E1 -21142.116,E2 -21142.116} C_VEL
LIN {X 0,Y 204.474,Z 391.956,A -85,B 0,C 180,E1 -21146.058,E2 -21146.058} C_VEL
LIN {X 0,Y 204.388,Z 392.639,A -85,B 0,C 180,E1 -21150,E2 -21150} C_VEL
LIN {X 0,Y 204.474,Z 392.009,A -85,B 0,C 180,E1 -21153.942,E2 -21153.942} C_VEL
LIN {X 0,Y 204.936,Z 390.049,A -85,B 0,C 180,E1 -21157.885,E2 -21157.885} C_VEL
LIN {X 0,Y 205.991,Z 386.71,A -85,B 0,C 180,E1 -21161.813,E2 -21161.813} C_VEL
LIN {X 0,Y 207.644,Z 381.894,A -85,B 0,C 180,E1 -21165.71,E2 -21165.71} C_VEL
LIN {X 0,Y 210.365,Z 375.436,A -85,B 0,C 180,E1 -21169.517,E2 -21169.517} C_VEL
LIN {X 0,Y 212.501,Z 369.364,A -85,B 0,C 180,E1 -21172.354,E2 -21172.354} C_VEL
LIN {X 0,Y 215.987,Z 360.71,A -85,B 0,C 180,E1 -21175.54,E2 -21175.54} C_VEL
LIN {X 0,Y 219.402,Z 351.653,A -85,B 0,C 180,E1 -21178.196,E2 -21178.196} C_VEL
LIN {X 0,Y 223.228,Z 340.677,A -85,B 0,C 180,E1 -21180.771,E2 -21180.771} C_VEL
LIN {X 0,Y 226.823,Z 329.141,A -85,B 0,C 180,E1 -21182.904,E2 -21182.904} C_VEL
LIN {X 0,Y 226.675,Z 322.731,A -85,B 0,C 180,E1 -21184.233,E2 -21184.233} C_VEL
LIN {X 0,Y 225.469,Z 312.445,A -85,B 0,C 180,E1 -21186.316,E2 -21186.316} C_VEL
LIN {X 0,Y 223.23,Z 301.206,A -85,B 0,C 180,E1 -21188.475,E2 -21188.475} C_VEL
LIN {X 0,Y 219.482,Z 288.789,A -85,B 0,C 180,E1 -21190.844,E2 -21190.844} C_VEL
LIN {X 0,Y 215.688,Z 279.869,A -85,B 0,C 180,E1 -21192.646,E2 -21192.646} C_VEL
LIN {X 0,Y 212.182,Z 272.872,A -85,B 0,C 180,E1 -21194.127,E2 -21194.127} C_VEL
LIN {X 0,Y 210.304,Z 269.464,A -85,B 0,C 180,E1 -21194.881,E2 -21194.881} C_VEL
LIN {X 0,Y 209.061,Z 267.688,A -85,B 0,C 180,E1 -21195.346,E2 -21195.346} C_VEL
LIN {X 0,Y 207.502,Z 264.865,A -85,B 0,C 180,E1 -21195.949,E2 -21195.949} C_VEL
LIN {X 0,Y 207.169,Z 263.648,A -85,B 0,C 180,E1 -21196.124,E2 -21196.124} C_VEL
LIN {X 0,Y 206.773,Z 261.007,A -85,B 0,C 180,E1 -21201.421,E2 -21201.421} C_VEL
LIN {X 0,Y 206.724,Z 260.609,A -85,B 0,C 180,E1 -21202.269,E2 -21202.269} C_VEL
LIN {X 0,Y 206.701,Z 260.365,A -85,B 0,C 180,E1 -21204.689,E2 -21204.689} C_VEL
LIN {X 0,Y 206.726,Z 260.36,A -85,B 0,C 180,E1 -21209.339,E2 -21209.339} C_VEL
LIN {X 0,Y 206.734,Z 260.357,A -85,B 0,C 180,E1 -21213.772,E2 -21213.772} C_VEL
LIN {X 0,Y 206.742,Z 260.357,A -85,B 0,C 180,E1 -21218.041,E2 -21218.041} C_VEL
LIN {X 0,Y 206.876,Z 260.34,A -85,B 0,C 180,E1 -21222.197,E2 -21222.197} C_VEL
LIN {X 0,Y 206.898,Z 260.337,A -85,B 0,C 180,E1 -21226.244,E2 -21226.244} C_VEL
LIN {X 0,Y 207.102,Z 260.313,A -85,B 0,C 180,E1 -21230.231,E2 -21230.231} C_VEL
LIN {X 0,Y 207.058,Z 260.316,A -85,B 0,C 180,E1 -21234.155,E2 -21234.155} C_VEL
LIN {X 0,Y 207.381,Z 260.277,A -85,B 0,C 180,E1 -21238.058,E2 -21238.058} C_VEL
LIN {X 0,Y 207.487,Z 260.263,A -85,B 0,C 180,E1 -21240,E2 -21240} C_VEL
LIN {X 0,Y 207.382,Z 260.276,A -85,B 0,C 180,E1 -21241.942,E2 -21241.942} C_VEL
LIN {X 0,Y 207.132,Z 260.307,A -85,B 0,C 180,E1 -21247.8,E2 -21247.8} C_VEL
LIN {X 0,Y 206.919,Z 260.335,A -85,B 0,C 180,E1 -21251.759,E2 -21251.759} C_VEL
LIN {X 0,Y 206.842,Z 260.347,A -85,B 0,C 180,E1 -21255.773,E2 -21255.773} C_VEL
LIN {X 0,Y 206.859,Z 260.345,A -85,B 0,C 180,E1 -21257.954,E2 -21257.954} C_VEL
LIN {X 0,Y 206.747,Z 260.357,A -85,B 0,C 180,E1 -21263.39,E2 -21263.39} C_VEL
LIN {X 0,Y 206.69,Z 260.363,A -85,B 0,C 180,E1 -21268.427,E2 -21268.427} C_VEL
LIN {X 0,Y 206.899,Z 261.543,A -85,B 0,C 180,E1 -21271.874,E2 -21271.874} C_VEL
LIN {X 0,Y 207.245,Z 263.483,A -85,B 0,C 180,E1 -21275.523,E2 -21275.523} C_VEL
LIN {X 0,Y 207.63,Z 266.139,A -85,B 0,C 180,E1 -21280.025,E2 -21280.025} C_VEL
LIN {X 0,Y 208.079,Z 268.961,A -85,B 0,C 180,E1 -21284.179,E2 -21284.179} C_VEL
LIN {X 0,Y 209.21,Z 271.997,A -85,B 0,C 180,E1 -21284.668,E2 -21284.668} C_VEL
LIN {X 0,Y 211.038,Z 274.619,A -85,B 0,C 180,E1 -21285.323,E2 -21285.323} C_VEL
LIN {X 0,Y 212.962,Z 278.44,A -85,B 0,C 180,E1 -21286.104,E2 -21286.104} C_VEL
LIN {X 0,Y 217.286,Z 288.301,A -85,B 0,C 180,E1 -21288,E2 -21288} C_VEL
LIN {X 0,Y 220.234,Z 297.379,A -85,B 0,C 180,E1 -21289.631,E2 -21289.631} C_VEL
LIN {X 0,Y 222.87,Z 308.54,A -85,B 0,C 180,E1 -21291.598,E2 -21291.598} C_VEL
LIN {X 0,Y 224.597,Z 320.269,A -85,B 0,C 180,E1 -21293.726,E2 -21293.726} C_VEL
LIN {X 0,Y 225.223,Z 332.676,A -85,B 0,C 180,E1 -21296.124,E2 -21296.124} C_VEL
LIN {X 0,Y 225.207,Z 338.153,A -85,B 0,C 180,E1 -21297.268,E2 -21297.268} C_VEL
LIN {X 0,Y 222.397,Z 347.765,A -85,B 0,C 180,E1 -21299.101,E2 -21299.101} C_VEL
LIN {X 0,Y 221.351,Z 350.783,A -85,B 0,C 180,E1 -21299.752,E2 -21299.752} C_VEL
LIN {X 0,Y 219.267,Z 355.097,A -85,B 0,C 180,E1 -21300.656,E2 -21300.656} C_VEL
LIN {X 0,Y 214.203,Z 361.813,A -85,B 0,C 180,E1 -21302.051,E2 -21302.051} C_VEL
LIN {X 0,Y 209.169,Z 368.044,A -85,B 0,C 180,E1 -21303.63,E2 -21303.63} C_VEL
LIN {X 0,Y 207.177,Z 371.574,A -85,B 0,C 180,E1 -21304.808,E2 -21304.808} C_VEL
LIN {X 0,Y 204.289,Z 378.779,A -85,B 0,C 180,E1 -21307.764,E2 -21307.764} C_VEL
LIN {X 0,Y 202.067,Z 384.548,A -85,B 0,C 180,E1 -21310.706,E2 -21310.706} C_VEL
LIN {X 0,Y 200.179,Z 389.27,A -85,B 0,C 180,E1 -21313.688,E2 -21313.688} C_VEL
LIN {X 0,Y 198.446,Z 394.169,A -85,B 0,C 180,E1 -21317.731,E2 -21317.731} C_VEL
LIN {X 0,Y 197.498,Z 397.578,A -85,B 0,C 180,E1 -21321.816,E2 -21321.816} C_VEL
LIN {X 0,Y 197.176,Z 399.596,A -85,B 0,C 180,E1 -21325.912,E2 -21325.912} C_VEL
LIN {X 0,Y 197.278,Z 400.262,A -85,B 0,C 180,E1 -21330,E2 -21330} C_VEL
LIN {X 0,Y 197.175,Z 399.577,A -85,B 0,C 180,E1 -21334.088,E2 -21334.088} C_VEL
LIN {X 0,Y 197.497,Z 397.544,A -85,B 0,C 180,E1 -21338.183,E2 -21338.183} C_VEL
LIN {X 0,Y 198.438,Z 394.116,A -85,B 0,C 180,E1 -21342.269,E2 -21342.269} C_VEL
LIN {X 0,Y 200.173,Z 389.193,A -85,B 0,C 180,E1 -21346.312,E2 -21346.312} C_VEL
LIN {X 0,Y 202.711,Z 382.631,A -85,B 0,C 180,E1 -21350.286,E2 -21350.286} C_VEL
LIN {X 0,Y 205.591,Z 375.333,A -85,B 0,C 180,E1 -21353.682,E2 -21353.682} C_VEL
LIN {X 0,Y 209.223,Z 366.296,A -85,B 0,C 180,E1 -21356.967,E2 -21356.967} C_VEL
LIN {X 0,Y 212.852,Z 356.82,A -85,B 0,C 180,E1 -21359.688,E2 -21359.688} C_VEL
LIN {X 0,Y 216.996,Z 345.348,A -85,B 0,C 180,E1 -21362.281,E2 -21362.281} C_VEL
LIN {X 0,Y 218.678,Z 339.961,A -85,B 0,C 180,E1 -21363.321,E2 -21363.321} C_VEL
LIN {X 0,Y 218.819,Z 330.768,A -85,B 0,C 180,E1 -21365.318,E2 -21365.318} C_VEL
LIN {X 0,Y 218.208,Z 319.724,A -85,B 0,C 180,E1 -21367.522,E2 -21367.522} C_VEL
LIN {X 0,Y 216.309,Z 307.443,A -85,B 0,C 180,E1 -21369.863,E2 -21369.863} C_VEL
LIN {X 0,Y 213.613,Z 296.592,A -85,B 0,C 180,E1 -21371.894,E2 -21371.894} C_VEL
LIN {X 0,Y 210.006,Z 286.702,A -85,B 0,C 180,E1 -21373.874,E2 -21373.874} C_VEL
LIN {X 0,Y 207.759,Z 281.965,A -85,B 0,C 180,E1 -21374.906,E2 -21374.906} C_VEL
LIN {X 0,Y 205.955,Z 278.365,A -85,B 0,C 180,E1 -21375.705,E2 -21375.705} C_VEL
LIN {X 0,Y 204.152,Z 274.951,A -85,B 0,C 180,E1 -21376.488,E2 -21376.488} C_VEL
LIN {X 0,Y 203.429,Z 273.684,A -85,B 0,C 180,E1 -21376.798,E2 -21376.798} C_VEL
LIN {X 0,Y 201.487,Z 270.783,A -85,B 0,C 180,E1 -21377.566,E2 -21377.566} C_VEL
LIN {X 0,Y 200.829,Z 268.594,A -85,B 0,C 180,E1 -21377.952,E2 -21377.952} C_VEL
LIN {X 0,Y 200.566,Z 266.796,A -85,B 0,C 180,E1 -21380.896,E2 -21380.896} C_VEL
LIN {X 0,Y 200.317,Z 265.164,A -85,B 0,C 180,E1 -21383.798,E2 -21383.798} C_VEL
LIN {X 0,Y 199.942,Z 262.885,A -85,B 0,C 180,E1 -21388.18,E2 -21388.18} C_VEL
LIN {X 0,Y 199.666,Z 261.244,A -85,B 0,C 180,E1 -21391.639,E2 -21391.639} C_VEL
LIN {X 0,Y 199.708,Z 261.234,A -85,B 0,C 180,E1 -21397.226,E2 -21397.226} C_VEL
LIN {X 0,Y 199.751,Z 261.224,A -85,B 0,C 180,E1 -21401.798,E2 -21401.798} C_VEL
LIN {X 0,Y 199.82,Z 261.213,A -85,B 0,C 180,E1 -21405.747,E2 -21405.747} C_VEL
LIN {X 0,Y 200.023,Z 261.186,A -85,B 0,C 180,E1 -21409.882,E2 -21409.882} C_VEL
LIN {X 0,Y 200.013,Z 261.196,A -85,B 0,C 180,E1 -21413.949,E2 -21413.949} C_VEL
LIN {X 0,Y 200.32,Z 261.158,A -85,B 0,C 180,E1 -21417.99,E2 -21417.99} C_VEL
LIN {X 0,Y 200.472,Z 261.138,A -85,B 0,C 180,E1 -21420,E2 -21420} C_VEL
LIN {X 0,Y 200.024,Z 261.192,A -85,B 0,C 180,E1 -21424.03,E2 -21424.03} C_VEL
LIN {X 0,Y 200.09,Z 261.187,A -85,B 0,C 180,E1 -21428.077,E2 -21428.077} C_VEL
LIN {X 0,Y 199.881,Z 261.212,A -85,B 0,C 180,E1 -21432.179,E2 -21432.179} C_VEL
LIN {X 0,Y 199.806,Z 261.221,A -85,B 0,C 180,E1 -21436.344,E2 -21436.344} C_VEL
LIN {X 0,Y 199.684,Z 261.236,A -85,B 0,C 180,E1 -21440.607,E2 -21440.607} C_VEL
LIN {X 0,Y 199.666,Z 261.239,A -85,B 0,C 180,E1 -21444.986,E2 -21444.986} C_VEL
LIN {X 0,Y 199.666,Z 261.237,A -85,B 0,C 180,E1 -21449.524,E2 -21449.524} C_VEL
LIN {X 0,Y 199.672,Z 261.238,A -85,B 0,C 180,E1 -21452.355,E2 -21452.355} C_VEL
LIN {X 0,Y 199.629,Z 261.469,A -85,B 0,C 180,E1 -21456.762,E2 -21456.762} C_VEL
LIN {X 0,Y 199.83,Z 262.605,A -85,B 0,C 180,E1 -21459.309,E2 -21459.309} C_VEL
LIN {X 0,Y 199.992,Z 263.83,A -85,B 0,C 180,E1 -21461.889,E2 -21461.889} C_VEL
LIN {X 0,Y 201.159,Z 266.842,A -85,B 0,C 180,E1 -21462.452,E2 -21462.452} C_VEL
LIN {X 0,Y 203.294,Z 269.618,A -85,B 0,C 180,E1 -21463.3,E2 -21463.3} C_VEL
LIN {X 0,Y 205.373,Z 273.335,A -85,B 0,C 180,E1 -21464.206,E2 -21464.206} C_VEL
LIN {X 0,Y 208.847,Z 279.841,A -85,B 0,C 180,E1 -21465.759,E2 -21465.759} C_VEL
LIN {X 0,Y 212.057,Z 286.931,A -85,B 0,C 180,E1 -21467.336,E2 -21467.336} C_VEL
LIN {X 0,Y 214.687,Z 294.144,A -85,B 0,C 180,E1 -21468.845,E2 -21468.845} C_VEL
LIN {X 0,Y 217.414,Z 304.111,A -85,B 0,C 180,E1 -21470.879,E2 -21470.879} C_VEL
LIN {X 0,Y 219.66,Z 316.893,A -85,B 0,C 180,E1 -21473.502,E2 -21473.502} C_VEL
LIN {X 0,Y 220.527,Z 328.22,A -85,B 0,C 180,E1 -21475.955,E2 -21475.955} C_VEL
LIN {X 0,Y 220.235,Z 331.106,A -85,B 0,C 180,E1 -21476.546,E2 -21476.546} C_VEL
LIN {X 0,Y 216.537,Z 342.221,A -85,B 0,C 180,E1 -21478.715,E2 -21478.715} C_VEL
LIN {X 0,Y 212.637,Z 352.958,A -85,B 0,C 180,E1 -21481.364,E2 -21481.364} C_VEL
LIN {X 0,Y 209.089,Z 361.817,A -85,B 0,C 180,E1 -21484.09,E2 -21484.09} C_VEL
LIN {X 0,Y 205.618,Z 370.216,A -85,B 0,C 180,E1 -21487.348,E2 -21487.348} C_VEL
LIN {X 0,Y 202.947,Z 377.117,A -85,B 0,C 180,E1 -21490.793,E2 -21490.793} C_VEL
LIN {X 0,Y 200.835,Z 381.827,A -85,B 0,C 180,E1 -21493.743,E2 -21493.743} C_VEL
LIN {X 0,Y 199.045,Z 386.699,A -85,B 0,C 180,E1 -21497.769,E2 -21497.769} C_VEL
LIN {X 0,Y 197.905,Z 390.086,A -85,B 0,C 180,E1 -21501.834,E2 -21501.834} C_VEL
LIN {X 0,Y 197.395,Z 392.091,A -85,B 0,C 180,E1 -21505.917,E2 -21505.917} C_VEL
LIN {X 0,Y 197.294,Z 392.773,A -85,B 0,C 180,E1 -21510,E2 -21510} C_VEL
LIN {X 0,Y 197.395,Z 392.143,A -85,B 0,C 180,E1 -21514.084,E2 -21514.084} C_VEL
LIN {X 0,Y 197.905,Z 390.183,A -85,B 0,C 180,E1 -21518.167,E2 -21518.167} C_VEL
LIN {X 0,Y 199.018,Z 386.844,A -85,B 0,C 180,E1 -21522.233,E2 -21522.233} C_VEL
LIN {X 0,Y 200.79,Z 382.028,A -85,B 0,C 180,E1 -21526.261,E2 -21526.261} C_VEL
LIN {X 0,Y 202.897,Z 377.37,A -85,B 0,C 180,E1 -21529.212,E2 -21529.212} C_VEL
LIN {X 0,Y 205.267,Z 371.105,A -85,B 0,C 180,E1 -21532.416,E2 -21532.416} C_VEL
LIN {X 0,Y 208.466,Z 363.539,A -85,B 0,C 180,E1 -21535.458,E2 -21535.458} C_VEL
LIN {X 0,Y 211.947,Z 355.026,A -85,B 0,C 180,E1 -21538.198,E2 -21538.198} C_VEL
LIN {X 0,Y 215.734,Z 344.705,A -85,B 0,C 180,E1 -21540.87,E2 -21540.87} C_VEL
LIN {X 0,Y 219.335,Z 334.326,A -85,B 0,C 180,E1 -21543.006,E2 -21543.006} C_VEL
LIN {X 0,Y 220.611,Z 329.956,A -85,B 0,C 180,E1 -21543.807,E2 -21543.807} C_VEL
LIN {X 0,Y 220.107,Z 320.526,A -85,B 0,C 180,E1 -21545.872,E2 -21545.872} C_VEL
LIN {X 0,Y 218.597,Z 309.718,A -85,B 0,C 180,E1 -21548.133,E2 -21548.133} C_VEL
LIN {X 0,Y 216.305,Z 299.441,A -85,B 0,C 180,E1 -21550.223,E2 -21550.223} C_VEL
LIN {X 0,Y 213.309,Z 290.051,A -85,B 0,C 180,E1 -21552.156,E2 -21552.156} C_VEL
LIN {X 0,Y 209.463,Z 281.041,A -85,B 0,C 180,E1 -21554.141,E2 -21554.141} C_VEL
LIN {X 0,Y 207.211,Z 276.772,A -85,B 0,C 180,E1 -21555.156,E2 -21555.156} C_VEL
LIN {X 0,Y 205.235,Z 273.164,A -85,B 0,C 180,E1 -21556.03,E2 -21556.03} C_VEL
LIN {X 0,Y 203.253,Z 269.47,A -85,B 0,C 180,E1 -21556.909,E2 -21556.909} C_VEL
LIN {X 0,Y 200.78,Z 266.204,A -85,B 0,C 180,E1 -21557.896,E2 -21557.896} C_VEL
LIN {X 0,Y 199.997,Z 263.803,A -85,B 0,C 180,E1 -21558.365,E2 -21558.365} C_VEL
LIN {X 0,Y 199.65,Z 261.562,A -85,B 0,C 180,E1 -21563.242,E2 -21563.242} C_VEL
LIN {X 0,Y 199.62,Z 261.245,A -85,B 0,C 180,E1 -21564.073,E2 -21564.073} C_VEL
LIN {X 0,Y 199.703,Z 261.235,A -85,B 0,C 180,E1 -21568.137,E2 -21568.137} C_VEL
LIN {X 0,Y 199.689,Z 261.236,A -85,B 0,C 180,E1 -21572.772,E2 -21572.772} C_VEL
LIN {X 0,Y 199.717,Z 261.233,A -85,B 0,C 180,E1 -21577.226,E2 -21577.226} C_VEL
LIN {X 0,Y 199.799,Z 261.221,A -85,B 0,C 180,E1 -21581.758,E2 -21581.758} C_VEL
LIN {X 0,Y 199.839,Z 261.218,A -85,B 0,C 180,E1 -21585.748,E2 -21585.748} C_VEL
LIN {X 0,Y 200.025,Z 261.193,A -85,B 0,C 180,E1 -21589.882,E2 -21589.882} C_VEL
LIN {X 0,Y 200.02,Z 261.193,A -85,B 0,C 180,E1 -21593.949,E2 -21593.949} C_VEL
LIN {X 0,Y 200.32,Z 261.156,A -85,B 0,C 180,E1 -21597.989,E2 -21597.989} C_VEL
LIN {X 0,Y 200.455,Z 261.138,A -85,B 0,C 180,E1 -21600,E2 -21600} C_VEL
LIN {X 0,Y 200.321,Z 261.155,A -85,B 0,C 180,E1 -21602.01,E2 -21602.01} C_VEL
LIN {X 0,Y 200.08,Z 261.187,A -85,B 0,C 180,E1 -21608.077,E2 -21608.077} C_VEL
LIN {X 0,Y 199.868,Z 261.212,A -85,B 0,C 180,E1 -21612.18,E2 -21612.18} C_VEL
LIN {X 0,Y 199.787,Z 261.224,A -85,B 0,C 180,E1 -21616.345,E2 -21616.345} C_VEL
LIN {X 0,Y 199.677,Z 261.237,A -85,B 0,C 180,E1 -21620.608,E2 -21620.608} C_VEL
LIN {X 0,Y 199.652,Z 261.234,A -85,B 0,C 180,E1 -21624.987,E2 -21624.987} C_VEL
LIN {X 0,Y 199.667,Z 261.311,A -85,B 0,C 180,E1 -21628.361,E2 -21628.361} C_VEL
LIN {X 0,Y 199.969,Z 263.285,A -85,B 0,C 180,E1 -21632.489,E2 -21632.489} C_VEL
LIN {X 0,Y 200.357,Z 265.444,A -85,B 0,C 180,E1 -21636.606,E2 -21636.606} C_VEL
LIN {X 0,Y 200.617,Z 267.138,A -85,B 0,C 180,E1 -21639.582,E2 -21639.582} C_VEL
LIN {X 0,Y 200.831,Z 268.628,A -85,B 0,C 180,E1 -21641.999,E2 -21641.999} C_VEL
LIN {X 0,Y 201.965,Z 271.723,A -85,B 0,C 180,E1 -21642.542,E2 -21642.542} C_VEL
LIN {X 0,Y 203.958,Z 274.381,A -85,B 0,C 180,E1 -21643.317,E2 -21643.317} C_VEL
LIN {X 0,Y 205.771,Z 278.1,A -85,B 0,C 180,E1 -21644.132,E2 -21644.132} C_VEL
LIN {X 0,Y 206.798,Z 279.775,A -85,B 0,C 180,E1 -21644.55,E2 -21644.55} C_VEL
LIN {X 0,Y 210.593,Z 288.001,A -85,B 0,C 180,E1 -21646.324,E2 -21646.324} C_VEL
LIN {X 0,Y 213.723,Z 296.75,A -85,B 0,C 180,E1 -21648.073,E2 -21648.073} C_VEL
LIN {X 0,Y 216.671,Z 309.049,A -85,B 0,C 180,E1 -21650.385,E2 -21650.385} C_VEL
LIN {X 0,Y 218.303,Z 320.314,A -85,B 0,C 180,E1 -21652.538,E2 -21652.538} C_VEL
LIN {X 0,Y 218.882,Z 331.081,A -85,B 0,C 180,E1 -21654.693,E2 -21654.693} C_VEL
LIN {X 0,Y 218.754,Z 340.037,A -85,B 0,C 180,E1 -21656.648,E2 -21656.648} C_VEL
LIN {X 0,Y 214.91,Z 351.554,A -85,B 0,C 180,E1 -21658.998,E2 -21658.998} C_VEL
LIN {X 0,Y 210.957,Z 361.961,A -85,B 0,C 180,E1 -21661.657,E2 -21661.657} C_VEL
LIN {X 0,Y 207.577,Z 370.553,A -85,B 0,C 180,E1 -21664.425,E2 -21664.425} C_VEL
LIN {X 0,Y 207.177,Z 371.574,A -85,B 0,C 180,E1 -21664.808,E2 -21664.808} C_VEL
LIN {X 0,Y 205.245,Z 374.972,A -85,B 0,C 180,E1 -21666.051,E2 -21666.051} C_VEL
LIN {X 0,Y 200.466,Z 380.066,A -85,B 0,C 180,E1 -21668.042,E2 -21668.042} C_VEL
LIN {X 0,Y 195.83,Z 384.661,A -85,B 0,C 180,E1 -21670.208,E2 -21670.208} C_VEL
LIN {X 0,Y 194.167,Z 387.128,A -85,B 0,C 180,E1 -21671.697,E2 -21671.697} C_VEL
LIN {X 0,Y 192.225,Z 391.779,A -85,B 0,C 180,E1 -21675.171,E2 -21675.171} C_VEL
LIN {X 0,Y 190.863,Z 395.918,A -85,B 0,C 180,E1 -21679.39,E2 -21679.39} C_VEL
LIN {X 0,Y 190.221,Z 398.623,A -85,B 0,C 180,E1 -21683.636,E2 -21683.636} C_VEL
LIN {X 0,Y 190.085,Z 399.962,A -85,B 0,C 180,E1 -21687.881,E2 -21687.881} C_VEL
LIN {X 0,Y 190.184,Z 400.127,A -85,B 0,C 180,E1 -21690,E2 -21690} C_VEL
LIN {X 0,Y 190.086,Z 399.442,A -85,B 0,C 180,E1 -21694.24,E2 -21694.24} C_VEL
LIN {X 0,Y 190.456,Z 397.409,A -85,B 0,C 180,E1 -21698.488,E2 -21698.488} C_VEL
LIN {X 0,Y 191.459,Z 393.98,A -85,B 0,C 180,E1 -21702.723,E2 -21702.723} C_VEL
LIN {X 0,Y 193.337,Z 389.057,A -85,B 0,C 180,E1 -21706.906,E2 -21706.906} C_VEL
LIN {X 0,Y 195.311,Z 384.313,A -85,B 0,C 180,E1 -21709.989,E2 -21709.989} C_VEL
LIN {X 0,Y 198.092,Z 377.437,A -85,B 0,C 180,E1 -21713.524,E2 -21713.524} C_VEL
LIN {X 0,Y 201.691,Z 368.909,A -85,B 0,C 180,E1 -21716.936,E2 -21716.936} C_VEL
LIN {X 0,Y 205.323,Z 360.014,A -85,B 0,C 180,E1 -21719.757,E2 -21719.757} C_VEL
LIN {X 0,Y 209.544,Z 349.246,A -85,B 0,C 180,E1 -21722.455,E2 -21722.455} C_VEL
LIN {X 0,Y 212.393,Z 340.693,A -85,B 0,C 180,E1 -21724.23,E2 -21724.23} C_VEL
LIN {X 0,Y 212.571,Z 329.947,A -85,B 0,C 180,E1 -21726.658,E2 -21726.658} C_VEL
LIN {X 0,Y 211.947,Z 319.687,A -85,B 0,C 180,E1 -21728.81,E2 -21728.81} C_VEL
LIN {X 0,Y 210.473,Z 309.663,A -85,B 0,C 180,E1 -21730.828,E2 -21730.828} C_VEL
LIN {X 0,Y 207.683,Z 298.027,A -85,B 0,C 180,E1 -21733.176,E2 -21733.176} C_VEL
LIN {X 0,Y 203.928,Z 287.899,A -85,B 0,C 180,E1 -21735.394,E2 -21735.394} C_VEL
LIN {X 0,Y 200.988,Z 282.135,A -85,B 0,C 180,E1 -21736.827,E2 -21736.827} C_VEL
LIN {X 0,Y 199.226,Z 278.658,A -85,B 0,C 180,E1 -21737.684,E2 -21737.684} C_VEL
LIN {X 0,Y 197.194,Z 275.033,A -85,B 0,C 180,E1 -21738.637,E2 -21738.637} C_VEL
LIN {X 0,Y 196.461,Z 273.682,A -85,B 0,C 180,E1 -21738.991,E2 -21738.991} C_VEL
LIN {X 0,Y 194.394,Z 270.844,A -85,B 0,C 180,E1 -21739.886,E2 -21739.886} C_VEL
LIN {X 0,Y 193.625,Z 268.384,A -85,B 0,C 180,E1 -21740.389,E2 -21740.389} C_VEL
LIN {X 0,Y 193.263,Z 266.196,A -85,B 0,C 180,E1 -21744.42,E2 -21744.42} C_VEL
LIN {X 0,Y 192.844,Z 263.766,A -85,B 0,C 180,E1 -21749.322,E2 -21749.322} C_VEL
LIN {X 0,Y 192.711,Z 262.69,A -85,B 0,C 180,E1 -21751.7,E2 -21751.7} C_VEL
LIN {X 0,Y 192.569,Z 262.124,A -85,B 0,C 180,E1 -21754.027,E2 -21754.027} C_VEL
LIN {X 0,Y 192.679,Z 262.111,A -85,B 0,C 180,E1 -21756.345,E2 -21756.345} C_VEL
LIN {X 0,Y 192.7,Z 262.104,A -85,B 0,C 180,E1 -21761.487,E2 -21761.487} C_VEL
LIN {X 0,Y 192.744,Z 262.095,A -85,B 0,C 180,E1 -21765.212,E2 -21765.212} C_VEL
LIN {X 0,Y 192.946,Z 262.067,A -85,B 0,C 180,E1 -21769.567,E2 -21769.567} C_VEL
LIN {X 0,Y 192.976,Z 262.073,A -85,B 0,C 180,E1 -21773.728,E2 -21773.728} C_VEL
LIN {X 0,Y 193.261,Z 262.037,A -85,B 0,C 180,E1 -21777.916,E2 -21777.916} C_VEL
LIN {X 0,Y 193.437,Z 262.014,A -85,B 0,C 180,E1 -21780,E2 -21780} C_VEL
LIN {X 0,Y 192.97,Z 262.071,A -85,B 0,C 180,E1 -21784.177,E2 -21784.177} C_VEL
LIN {X 0,Y 193.038,Z 262.064,A -85,B 0,C 180,E1 -21788.374,E2 -21788.374} C_VEL
LIN {X 0,Y 192.807,Z 262.094,A -85,B 0,C 180,E1 -21792.633,E2 -21792.633} C_VEL
LIN {X 0,Y 192.759,Z 262.1,A -85,B 0,C 180,E1 -21796.959,E2 -21796.959} C_VEL
LIN {X 0,Y 192.618,Z 262.117,A -85,B 0,C 180,E1 -21801.4,E2 -21801.4} C_VEL
LIN {X 0,Y 192.649,Z 262.111,A -85,B 0,C 180,E1 -21804.214,E2 -21804.214} C_VEL
LIN {X 0,Y 192.645,Z 262.113,A -85,B 0,C 180,E1 -21808.889,E2 -21808.889} C_VEL
LIN {X 0,Y 192.597,Z 262.119,A -85,B 0,C 180,E1 -21813.186,E2 -21813.186} C_VEL
LIN {X 0,Y 192.626,Z 262.424,A -85,B 0,C 180,E1 -21815.716,E2 -21815.716} C_VEL
LIN {X 0,Y 192.9,Z 264.211,A -85,B 0,C 180,E1 -21819.499,E2 -21819.499} C_VEL
LIN {X 0,Y 194.072,Z 267.155,A -85,B 0,C 180,E1 -21820.118,E2 -21820.118} C_VEL
LIN {X 0,Y 196.335,Z 269.966,A -85,B 0,C 180,E1 -21821.111,E2 -21821.111} C_VEL
LIN {X 0,Y 198.244,Z 273.436,A -85,B 0,C 180,E1 -21822.035,E2 -21822.035} C_VEL
LIN {X 0,Y 199.495,Z 275.28,A -85,B 0,C 180,E1 -21822.59,E2 -21822.59} C_VEL
LIN {X 0,Y 204.222,Z 284.364,A -85,B 0,C 180,E1 -21824.955,E2 -21824.955} C_VEL
LIN {X 0,Y 208.303,Z 294.232,A -85,B 0,C 180,E1 -21827.281,E2 -21827.281} C_VEL
LIN {X 0,Y 211.501,Z 306.026,A -85,B 0,C 180,E1 -21829.843,E2 -21829.843} C_VEL
LIN {X 0,Y 213.323,Z 317.144,A -85,B 0,C 180,E1 -21832.25,E2 -21832.25} C_VEL
LIN {X 0,Y 214.166,Z 327.184,A -85,B 0,C 180,E1 -21834.53,E2 -21834.53} C_VEL
LIN {X 0,Y 214.293,Z 330.39,A -85,B 0,C 180,E1 -21835.28,E2 -21835.28} C_VEL
LIN {X 0,Y 213.5,Z 333.818,A -85,B 0,C 180,E1 -21835.972,E2 -21835.972} C_VEL
LIN {X 0,Y 209.781,Z 344.305,A -85,B 0,C 180,E1 -21838.153,E2 -21838.153} C_VEL
LIN {X 0,Y 205.789,Z 354.717,A -85,B 0,C 180,E1 -21840.879,E2 -21840.879} C_VEL
LIN {X 0,Y 202.143,Z 363.303,A -85,B 0,C 180,E1 -21843.686,E2 -21843.686} C_VEL
LIN {X 0,Y 198.579,Z 371.527,A -85,B 0,C 180,E1 -21847.089,E2 -21847.089} C_VEL
LIN {X 0,Y 196.241,Z 377.254,A -85,B 0,C 180,E1 -21850.11,E2 -21850.11} C_VEL
LIN {X 0,Y 194.007,Z 381.964,A -85,B 0,C 180,E1 -21853.154,E2 -21853.154} C_VEL
LIN {X 0,Y 192.094,Z 386.835,A -85,B 0,C 180,E1 -21857.319,E2 -21857.319} C_VEL
LIN {X 0,Y 190.857,Z 390.221,A -85,B 0,C 180,E1 -21861.53,E2 -21861.53} C_VEL
LIN {X 0,Y 190.317,Z 392.226,A -85,B 0,C 180,E1 -21865.765,E2 -21865.765} C_VEL
LIN {X 0,Y 190.201,Z 392.908,A -85,B 0,C 180,E1 -21870,E2 -21870} C_VEL
LIN {X 0,Y 190.331,Z 392.2,A -85,B 0,C 180,E1 -21874.45,E2 -21874.45} C_VEL
LIN {X 0,Y 190.856,Z 390.317,A -85,B 0,C 180,E1 -21878.47,E2 -21878.47} C_VEL
LIN {X 0,Y 192.07,Z 386.979,A -85,B 0,C 180,E1 -21882.683,E2 -21882.683} C_VEL
LIN {X 0,Y 193.964,Z 382.162,A -85,B 0,C 180,E1 -21886.85,E2 -21886.85} C_VEL
LIN {X 0,Y 196.183,Z 377.504,A -85,B 0,C 180,E1 -21889.897,E2 -21889.897} C_VEL
LIN {X 0,Y 198.549,Z 371.602,A -85,B 0,C 180,E1 -21893.027,E2 -21893.027} C_VEL
LIN {X 0,Y 202.058,Z 363.672,A -85,B 0,C 180,E1 -21896.326,E2 -21896.326} C_VEL
LIN {X 0,Y 205.707,Z 355.158,A -85,B 0,C 180,E1 -21899.134,E2 -21899.134} C_VEL
LIN {X 0,Y 209.655,Z 344.837,A -85,B 0,C 180,E1 -21901.869,E2 -21901.869} C_VEL
LIN {X 0,Y 213.419,Z 334.456,A -85,B 0,C 180,E1 -21904.044,E2 -21904.044} C_VEL
LIN {X 0,Y 214.308,Z 331.555,A -85,B 0,C 180,E1 -21904.587,E2 -21904.587} C_VEL
LIN {X 0,Y 213.944,Z 321.927,A -85,B 0,C 180,E1 -21906.813,E2 -21906.813} C_VEL
LIN {X 0,Y 212.501,Z 311.049,A -85,B 0,C 180,E1 -21909.227,E2 -21909.227} C_VEL
LIN {X 0,Y 210.767,Z 302.719,A -85,B 0,C 180,E1 -21911.025,E2 -21911.025} C_VEL
LIN {X 0,Y 208.025,Z 293.472,A -85,B 0,C 180,E1 -21913.064,E2 -21913.064} C_VEL
LIN {X 0,Y 204.556,Z 285.089,A -85,B 0,C 180,E1 -21915.048,E2 -21915.048} C_VEL
LIN {X 0,Y 200.812,Z 277.808,A -85,B 0,C 180,E1 -21916.934,E2 -21916.934} C_VEL
LIN {X 0,Y 198.649,Z 273.939,A -85,B 0,C 180,E1 -21917.985,E2 -21917.985} C_VEL
LIN {X 0,Y 196.491,Z 270.412,A -85,B 0,C 180,E1 -21918.995,E2 -21918.995} C_VEL
LIN {X 0,Y 195.813,Z 269.168,A -85,B 0,C 180,E1 -21919.333,E2 -21919.333} C_VEL
LIN {X 0,Y 193.696,Z 266.421,A -85,B 0,C 180,E1 -21920.267,E2 -21920.267} C_VEL
LIN {X 0,Y 192.86,Z 264.011,A -85,B 0,C 180,E1 -21920.78,E2 -21920.78} C_VEL
LIN {X 0,Y 192.632,Z 262.521,A -85,B 0,C 180,E1 -21924.285,E2 -21924.285} C_VEL
LIN {X 0,Y 192.613,Z 262.119,A -85,B 0,C 180,E1 -21927.058,E2 -21927.058} C_VEL
LIN {X 0,Y 192.667,Z 262.112,A -85,B 0,C 180,E1 -21931.692,E2 -21931.692} C_VEL
LIN {X 0,Y 192.688,Z 262.107,A -85,B 0,C 180,E1 -21936.346,E2 -21936.346} C_VEL
LIN {X 0,Y 192.734,Z 262.102,A -85,B 0,C 180,E1 -21941.458,E2 -21941.458} C_VEL
LIN {X 0,Y 192.767,Z 262.098,A -85,B 0,C 180,E1 -21945.214,E2 -21945.214} C_VEL
LIN {X 0,Y 192.948,Z 262.073,A -85,B 0,C 180,E1 -21949.567,E2 -21949.567} C_VEL
LIN {X 0,Y 192.983,Z 262.071,A -85,B 0,C 180,E1 -21953.728,E2 -21953.728} C_VEL
LIN {X 0,Y 193.262,Z 262.035,A -85,B 0,C 180,E1 -21957.916,E2 -21957.916} C_VEL
LIN {X 0,Y 193.422,Z 262.014,A -85,B 0,C 180,E1 -21960,E2 -21960} C_VEL
LIN {X 0,Y 192.967,Z 262.074,A -85,B 0,C 180,E1 -21964.177,E2 -21964.177} C_VEL
LIN {X 0,Y 193.03,Z 262.066,A -85,B 0,C 180,E1 -21968.374,E2 -21968.374} C_VEL
LIN {X 0,Y 192.795,Z 262.094,A -85,B 0,C 180,E1 -21972.634,E2 -21972.634} C_VEL
LIN {X 0,Y 192.747,Z 262.1,A -85,B 0,C 180,E1 -21976.96,E2 -21976.96} C_VEL
LIN {X 0,Y 192.612,Z 262.117,A -85,B 0,C 180,E1 -21981.4,E2 -21981.4} C_VEL
LIN {X 0,Y 192.641,Z 262.113,A -85,B 0,C 180,E1 -21984.208,E2 -21984.208} C_VEL
LIN {X 0,Y 192.57,Z 262.114,A -85,B 0,C 180,E1 -21985.973,E2 -21985.973} C_VEL
LIN {X 0,Y 192.726,Z 263.037,A -85,B 0,C 180,E1 -21988.932,E2 -21988.932} C_VEL
LIN {X 0,Y 193.053,Z 265.023,A -85,B 0,C 180,E1 -21993.143,E2 -21993.143} C_VEL
LIN {X 0,Y 193.475,Z 267.625,A -85,B 0,C 180,E1 -21998.136,E2 -21998.136} C_VEL
LIN {X 0,Y 193.672,Z 268.636,A -85,B 0,C 180,E1 -21999.602,E2 -21999.602} C_VEL
LIN {X 0,Y 194.889,Z 271.736,A -85,B 0,C 180,E1 -22000.236,E2 -22000.236} C_VEL
LIN {X 0,Y 197.058,Z 274.605,A -85,B 0,C 180,E1 -22001.179,E2 -22001.179} C_VEL
LIN {X 0,Y 199.04,Z 278.386,A -85,B 0,C 180,E1 -22002.135,E2 -22002.135} C_VEL
LIN {X 0,Y 200.216,Z 280.421,A -85,B 0,C 180,E1 -22002.671,E2 -22002.671} C_VEL
LIN {X 0,Y 204.184,Z 288.372,A -85,B 0,C 180,E1 -22004.642,E2 -22004.642} C_VEL
LIN {X 0,Y 207.649,Z 297.723,A -85,B 0,C 180,E1 -22006.692,E2 -22006.692} C_VEL
LIN {X 0,Y 210.213,Z 308.079,A -85,B 0,C 180,E1 -22008.783,E2 -22008.783} C_VEL
LIN {X 0,Y 211.912,Z 318.747,A -85,B 0,C 180,E1 -22010.94,E2 -22010.94} C_VEL
LIN {X 0,Y 212.606,Z 328.668,A -85,B 0,C 180,E1 -22013.018,E2 -22013.018} C_VEL
LIN {X 0,Y 212.558,Z 339.779,A -85,B 0,C 180,E1 -22015.513,E2 -22015.513} C_VEL
LIN {X 0,Y 211.854,Z 343.004,A -85,B 0,C 180,E1 -22016.185,E2 -22016.185} C_VEL
LIN {X 0,Y 208.117,Z 353.312,A -85,B 0,C 180,E1 -22018.437,E2 -22018.437} C_VEL
LIN {X 0,Y 204.05,Z 363.344,A -85,B 0,C 180,E1 -22021.171,E2 -22021.171} C_VEL
LIN {X 0,Y 200.476,Z 372.01,A -85,B 0,C 180,E1 -22024.158,E2 -22024.158} C_VEL
LIN {X 0,Y 197.214,Z 379.744,A -85,B 0,C 180,E1 -22027.522,E2 -22027.522} C_VEL
LIN {X 0,Y 194.589,Z 386.082,A -85,B 0,C 180,E1 -22031.031,E2 -22031.031} C_VEL
LIN {X 0,Y 194.167,Z 387.128,A -85,B 0,C 180,E1 -22031.697,E2 -22031.697} C_VEL
LIN {X 0,Y 192.602,Z 389.447,A -85,B 0,C 180,E1 -22033.238,E2 -22033.238} C_VEL
LIN {X 0,Y 188.489,Z 392.697,A -85,B 0,C 180,E1 -22035.769,E2 -22035.769} C_VEL
LIN {X 0,Y 185.276,Z 394.863,A -85,B 0,C 180,E1 -22037.906,E2 -22037.906} C_VEL
LIN {X 0,Y 183.774,Z 396.278,A -85,B 0,C 180,E1 -22039.635,E2 -22039.635} C_VEL
LIN {X 0,Y 183.566,Z 396.651,A -85,B 0,C 180,E1 -22040.233,E2 -22040.233} C_VEL
LIN {X 0,Y 183.137,Z 398.488,A -85,B 0,C 180,E1 -22043.389,E2 -22043.389} C_VEL
LIN {X 0,Y 182.991,Z 399.827,A -85,B 0,C 180,E1 -22047.799,E2 -22047.799} C_VEL
LIN {X 0,Y 183.092,Z 399.993,A -85,B 0,C 180,E1 -22050,E2 -22050} C_VEL
LIN {X 0,Y 183.014,Z 399.307,A -85,B 0,C 180,E1 -22054.405,E2 -22054.405} C_VEL
LIN {X 0,Y 183.405,Z 397.273,A -85,B 0,C 180,E1 -22058.817,E2 -22058.817} C_VEL
LIN {X 0,Y 184.478,Z 393.843,A -85,B 0,C 180,E1 -22063.213,E2 -22063.213} C_VEL
LIN {X 0,Y 186.523,Z 388.92,A -85,B 0,C 180,E1 -22067.544,E2 -22067.544} C_VEL
LIN {X 0,Y 188.594,Z 384.175,A -85,B 0,C 180,E1 -22070.733,E2 -22070.733} C_VEL
LIN {X 0,Y 191.559,Z 377.299,A -85,B 0,C 180,E1 -22074.377,E2 -22074.377} C_VEL
LIN {X 0,Y 195.366,Z 368.772,A -85,B 0,C 180,E1 -22077.882,E2 -22077.882} C_VEL
LIN {X 0,Y 199.173,Z 359.877,A -85,B 0,C 180,E1 -22080.773,E2 -22080.773} C_VEL
LIN {X 0,Y 203.575,Z 349.108,A -85,B 0,C 180,E1 -22083.529,E2 -22083.529} C_VEL
LIN {X 0,Y 206.112,Z 341.915,A -85,B 0,C 180,E1 -22085.08,E2 -22085.08} C_VEL
LIN {X 0,Y 206.415,Z 331.22,A -85,B 0,C 180,E1 -22087.629,E2 -22087.629} C_VEL
LIN {X 0,Y 206.102,Z 323.252,A -85,B 0,C 180,E1 -22089.39,E2 -22089.39} C_VEL
LIN {X 0,Y 204.935,Z 313.185,A -85,B 0,C 180,E1 -22091.569,E2 -22091.569} C_VEL
LIN {X 0,Y 202.574,Z 302.189,A -85,B 0,C 180,E1 -22093.937,E2 -22093.937} C_VEL
LIN {X 0,Y 199.167,Z 292.276,A -85,B 0,C 180,E1 -22096.259,E2 -22096.259} C_VEL
LIN {X 0,Y 195.19,Z 283.865,A -85,B 0,C 180,E1 -22098.471,E2 -22098.471} C_VEL
LIN {X 0,Y 193.012,Z 279.613,A -85,B 0,C 180,E1 -22099.651,E2 -22099.651} C_VEL
LIN {X 0,Y 190.416,Z 275.53,A -85,B 0,C 180,E1 -22100.944,E2 -22100.944} C_VEL
LIN {X 0,Y 189.588,Z 273.766,A -85,B 0,C 180,E1 -22101.414,E2 -22101.414} C_VEL
LIN {X 0,Y 187.475,Z 271.148,A -85,B 0,C 180,E1 -22102.426,E2 -22102.426} C_VEL
LIN {X 0,Y 186.452,Z 268.227,A -85,B 0,C 180,E1 -22103.077,E2 -22103.077} C_VEL
LIN {X 0,Y 185.964,Z 265.78,A -85,B 0,C 180,E1 -22108.056,E2 -22108.056} C_VEL
LIN {X 0,Y 185.632,Z 263.652,A -85,B 0,C 180,E1 -22112.979,E2 -22112.979} C_VEL
LIN {X 0,Y 185.581,Z 262.995,A -85,B 0,C 180,E1 -22115.382,E2 -22115.382} C_VEL
LIN {X 0,Y 185.635,Z 262.986,A -85,B 0,C 180,E1 -22121.17,E2 -22121.17} C_VEL
LIN {X 0,Y 185.673,Z 262.979,A -85,B 0,C 180,E1 -22124.636,E2 -22124.636} C_VEL
LIN {X 0,Y 185.889,Z 262.946,A -85,B 0,C 180,E1 -22129.419,E2 -22129.419} C_VEL
LIN {X 0,Y 185.939,Z 262.95,A -85,B 0,C 180,E1 -22133.489,E2 -22133.489} C_VEL
LIN {X 0,Y 186.205,Z 262.916,A -85,B 0,C 180,E1 -22137.837,E2 -22137.837} C_VEL
LIN {X 0,Y 186.401,Z 262.89,A -85,B 0,C 180,E1 -22140,E2 -22140} C_VEL
LIN {X 0,Y 185.917,Z 262.949,A -85,B 0,C 180,E1 -22144.336,E2 -22144.336} C_VEL
LIN {X 0,Y 185.985,Z 262.942,A -85,B 0,C 180,E1 -22148.694,E2 -22148.694} C_VEL
LIN {X 0,Y 185.733,Z 262.974,A -85,B 0,C 180,E1 -22153.123,E2 -22153.123} C_VEL
LIN {X 0,Y 185.691,Z 262.979,A -85,B 0,C 180,E1 -22157.625,E2 -22157.625} C_VEL
LIN {X 0,Y 185.58,Z 262.992,A -85,B 0,C 180,E1 -22162.254,E2 -22162.254} C_VEL
LIN {X 0,Y 185.56,Z 262.996,A -85,B 0,C 180,E1 -22167.033,E2 -22167.033} C_VEL
LIN {X 0,Y 185.578,Z 262.992,A -85,B 0,C 180,E1 -22169.493,E2 -22169.493} C_VEL
LIN {X 0,Y 185.537,Z 263.02,A -85,B 0,C 180,E1 -22173.556,E2 -22173.556} C_VEL
LIN {X 0,Y 185.702,Z 264.213,A -85,B 0,C 180,E1 -22176.673,E2 -22176.673} C_VEL
LIN {X 0,Y 186.881,Z 267.229,A -85,B 0,C 180,E1 -22177.412,E2 -22177.412} C_VEL
LIN {X 0,Y 189.43,Z 270.404,A -85,B 0,C 180,E1 -22178.676,E2 -22178.676} C_VEL
LIN {X 0,Y 191.486,Z 274.019,A -85,B 0,C 180,E1 -22179.774,E2 -22179.774} C_VEL
LIN {X 0,Y 192.661,Z 275.708,A -85,B 0,C 180,E1 -22180.353,E2 -22180.353} C_VEL
LIN {X 0,Y 195.935,Z 281.61,A -85,B 0,C 180,E1 -22182.103,E2 -22182.103} C_VEL
LIN {X 0,Y 198.667,Z 286.906,A -85,B 0,C 180,E1 -22183.617,E2 -22183.617} C_VEL
LIN {X 0,Y 202.855,Z 297.402,A -85,B 0,C 180,E1 -22186.3,E2 -22186.3} C_VEL
LIN {X 0,Y 205.603,Z 308.02,A -85,B 0,C 180,E1 -22188.765,E2 -22188.765} C_VEL
LIN {X 0,Y 207.259,Z 318.859,A -85,B 0,C 180,E1 -22191.253,E2 -22191.253} C_VEL
LIN {X 0,Y 207.938,Z 327.791,A -85,B 0,C 180,E1 -22193.405,E2 -22193.405} C_VEL
LIN {X 0,Y 208.015,Z 332.436,A -85,B 0,C 180,E1 -22194.559,E2 -22194.559} C_VEL
LIN {X 0,Y 205.301,Z 340.512,A -85,B 0,C 180,E1 -22196.201,E2 -22196.201} C_VEL
LIN {X 0,Y 201.648,Z 349.908,A -85,B 0,C 180,E1 -22198.48,E2 -22198.48} C_VEL
LIN {X 0,Y 197.685,Z 359.348,A -85,B 0,C 180,E1 -22201.318,E2 -22201.318} C_VEL
LIN {X 0,Y 193.523,Z 368.35,A -85,B 0,C 180,E1 -22204.742,E2 -22204.742} C_VEL
LIN {X 0,Y 190.334,Z 375.592,A -85,B 0,C 180,E1 -22208.331,E2 -22208.331} C_VEL
LIN {X 0,Y 187.955,Z 380.664,A -85,B 0,C 180,E1 -22211.468,E2 -22211.468} C_VEL
LIN {X 0,Y 186.08,Z 384.729,A -85,B 0,C 180,E1 -22214.67,E2 -22214.67} C_VEL
LIN {X 0,Y 184.409,Z 388.842,A -85,B 0,C 180,E1 -22219.015,E2 -22219.015} C_VEL
LIN {X 0,Y 183.449,Z 391.527,A -85,B 0,C 180,E1 -22223.401,E2 -22223.401} C_VEL
LIN {X 0,Y 183.107,Z 392.866,A -85,B 0,C 180,E1 -22227.801,E2 -22227.801} C_VEL
LIN {X 0,Y 183.111,Z 393.042,A -85,B 0,C 180,E1 -22230,E2 -22230} C_VEL
LIN {X 0,Y 183.232,Z 392.412,A -85,B 0,C 180,E1 -22234.4,E2 -22234.4} C_VEL
LIN {X 0,Y 183.82,Z 390.452,A -85,B 0,C 180,E1 -22238.797,E2 -22238.797} C_VEL
LIN {X 0,Y 185.14,Z 387.113,A -85,B 0,C 180,E1 -22243.166,E2 -22243.166} C_VEL
LIN {X 0,Y 187.166,Z 382.296,A -85,B 0,C 180,E1 -22247.482,E2 -22247.482} C_VEL
LIN {X 0,Y 189.495,Z 377.638,A -85,B 0,C 180,E1 -22250.631,E2 -22250.631} C_VEL
LIN {X 0,Y 192.416,Z 370.872,A -85,B 0,C 180,E1 -22254.262,E2 -22254.262} C_VEL
LIN {X 0,Y 196.324,Z 362.457,A -85,B 0,C 180,E1 -22257.735,E2 -22257.735} C_VEL
LIN {X 0,Y 200.168,Z 353.672,A -85,B 0,C 180,E1 -22260.604,E2 -22260.604} C_VEL
LIN {X 0,Y 204.437,Z 343.023,A -85,B 0,C 180,E1 -22263.37,E2 -22263.37} C_VEL
LIN {X 0,Y 208.104,Z 332.818,A -85,B 0,C 180,E1 -22265.486,E2 -22265.486} C_VEL
LIN {X 0,Y 207.73,Z 322.253,A -85,B 0,C 180,E1 -22268.067,E2 -22268.067} C_VEL
LIN {X 0,Y 206.259,Z 310.969,A -85,B 0,C 180,E1 -22270.699,E2 -22270.699} C_VEL
LIN {X 0,Y 203.895,Z 300.642,A -85,B 0,C 180,E1 -22273.105,E2 -22273.105} C_VEL
LIN {X 0,Y 200.485,Z 290.967,A -85,B 0,C 180,E1 -22275.484,E2 -22275.484} C_VEL
LIN {X 0,Y 196.589,Z 282.787,A -85,B 0,C 180,E1 -22277.737,E2 -22277.737} C_VEL
LIN {X 0,Y 194.421,Z 278.854,A -85,B 0,C 180,E1 -22278.894,E2 -22278.894} C_VEL
LIN {X 0,Y 191.935,Z 274.477,A -85,B 0,C 180,E1 -22280.227,E2 -22280.227} C_VEL
LIN {X 0,Y 189.781,Z 271.217,A -85,B 0,C 180,E1 -22281.324,E2 -22281.324} C_VEL
LIN {X 0,Y 188.94,Z 269.583,A -85,B 0,C 180,E1 -22281.8,E2 -22281.8} C_VEL
LIN {X 0,Y 186.695,Z 266.921,A -85,B 0,C 180,E1 -22282.904,E2 -22282.904} C_VEL
LIN {X 0,Y 185.718,Z 264.203,A -85,B 0,C 180,E1 -22283.583,E2 -22283.583} C_VEL
LIN {X 0,Y 185.564,Z 263.116,A -85,B 0,C 180,E1 -22286.432,E2 -22286.432} C_VEL
LIN {X 0,Y 185.584,Z 262.993,A -85,B 0,C 180,E1 -22290.576,E2 -22290.576} C_VEL
LIN {X 0,Y 185.582,Z 262.986,A -85,B 0,C 180,E1 -22295.382,E2 -22295.382} C_VEL
LIN {X 0,Y 185.676,Z 262.982,A -85,B 0,C 180,E1 -22301.134,E2 -22301.134} C_VEL
LIN {X 0,Y 185.698,Z 262.977,A -85,B 0,C 180,E1 -22304.637,E2 -22304.637} C_VEL
LIN {X 0,Y 185.891,Z 262.952,A -85,B 0,C 180,E1 -22309.418,E2 -22309.418} C_VEL
LIN {X 0,Y 185.946,Z 262.948,A -85,B 0,C 180,E1 -22313.489,E2 -22313.489} C_VEL
LIN {X 0,Y 186.206,Z 262.914,A -85,B 0,C 180,E1 -22317.837,E2 -22317.837} C_VEL
LIN {X 0,Y 186.388,Z 262.89,A -85,B 0,C 180,E1 -22320,E2 -22320} C_VEL
LIN {X 0,Y 185.914,Z 262.952,A -85,B 0,C 180,E1 -22324.336,E2 -22324.336} C_VEL
LIN {X 0,Y 185.978,Z 262.945,A -85,B 0,C 180,E1 -22328.694,E2 -22328.694} C_VEL
LIN {X 0,Y 185.722,Z 262.977,A -85,B 0,C 180,E1 -22333.123,E2 -22333.123} C_VEL
LIN {X 0,Y 185.685,Z 262.982,A -85,B 0,C 180,E1 -22337.625,E2 -22337.625} C_VEL
LIN {X 0,Y 185.574,Z 262.995,A -85,B 0,C 180,E1 -22342.254,E2 -22342.254} C_VEL
LIN {X 0,Y 185.579,Z 262.988,A -85,B 0,C 180,E1 -22344.646,E2 -22344.646} C_VEL
LIN {X 0,Y 185.805,Z 264.762,A -85,B 0,C 180,E1 -22349.545,E2 -22349.545} C_VEL
LIN {X 0,Y 186.174,Z 267.07,A -85,B 0,C 180,E1 -22354.489,E2 -22354.489} C_VEL
LIN {X 0,Y 186.459,Z 268.376,A -85,B 0,C 180,E1 -22356.837,E2 -22356.837} C_VEL
LIN {X 0,Y 187.641,Z 271.44,A -85,B 0,C 180,E1 -22357.537,E2 -22357.537} C_VEL
LIN {X 0,Y 190.053,Z 274.531,A -85,B 0,C 180,E1 -22358.713,E2 -22358.713} C_VEL
LIN {X 0,Y 192.004,Z 278.27,A -85,B 0,C 180,E1 -22359.765,E2 -22359.765} C_VEL
LIN {X 0,Y 193.227,Z 280.062,A -85,B 0,C 180,E1 -22360.355,E2 -22360.355} C_VEL
LIN {X 0,Y 196.485,Z 286.475,A -85,B 0,C 180,E1 -22362.118,E2 -22362.118} C_VEL
LIN {X 0,Y 198.993,Z 291.73,A -85,B 0,C 180,E1 -22363.527,E2 -22363.527} C_VEL
LIN {X 0,Y 202.489,Z 301.549,A -85,B 0,C 180,E1 -22365.854,E2 -22365.854} C_VEL
LIN {X 0,Y 204.737,Z 311.784,A -85,B 0,C 180,E1 -22368.063,E2 -22368.063} C_VEL
LIN {X 0,Y 206.011,Z 321.353,A -85,B 0,C 180,E1 -22370.136,E2 -22370.136} C_VEL
LIN {X 0,Y 206.495,Z 332.121,A -85,B 0,C 180,E1 -22372.528,E2 -22372.528} C_VEL
LIN {X 0,Y 206.192,Z 342.003,A -85,B 0,C 180,E1 -22374.888,E2 -22374.888} C_VEL
LIN {X 0,Y 202.086,Z 353.179,A -85,B 0,C 180,E1 -22377.381,E2 -22377.381} C_VEL
LIN {X 0,Y 197.824,Z 363.211,A -85,B 0,C 180,E1 -22380.173,E2 -22380.173} C_VEL
LIN {X 0,Y 194.205,Z 371.548,A -85,B 0,C 180,E1 -22383.105,E2 -22383.105} C_VEL
LIN {X 0,Y 190.607,Z 379.624,A -85,B 0,C 180,E1 -22386.706,E2 -22386.706} C_VEL
LIN {X 0,Y 187.853,Z 385.948,A -85,B 0,C 180,E1 -22390.323,E2 -22390.323} C_VEL
LIN {X 0,Y 185.34,Z 391.644,A -85,B 0,C 180,E1 -22394.607,E2 -22394.607} C_VEL
LIN {X 0,Y 183.854,Z 395.783,A -85,B 0,C 180,E1 -22398.981,E2 -22398.981} C_VEL
LIN {X 0,Y 183.566,Z 396.651,A -85,B 0,C 180,E1 -22400.233,E2 -22400.233} C_VEL
LIN {X 0,Y 182.594,Z 397.798,A -85,B 0,C 180,E1 -22402.022,E2 -22402.022} C_VEL
LIN {X 0,Y 179.422,Z 399.066,A -85,B 0,C 180,E1 -22404.969,E2 -22404.969} C_VEL
LIN {X 0,Y 176.951,Z 399.65,A -85,B 0,C 180,E1 -22407.41,E2 -22407.41} C_VEL
LIN {X 0,Y 176.017,Z 399.819,A -85,B 0,C 180,E1 -22409.319,E2 -22409.319} C_VEL
LIN {X 0,Y 175.999,Z 399.856,A -85,B 0,C 180,E1 -22409.965,E2 -22409.965} C_VEL
LIN {X 0,Y 175.935,Z 399.172,A -85,B 0,C 180,E1 -22414.582,E2 -22414.582} C_VEL
LIN {X 0,Y 176.351,Z 397.137,A -85,B 0,C 180,E1 -22419.172,E2 -22419.172} C_VEL
LIN {X 0,Y 177.515,Z 393.706,A -85,B 0,C 180,E1 -22423.742,E2 -22423.742} C_VEL
LIN {X 0,Y 179.714,Z 388.783,A -85,B 0,C 180,E1 -22428.231,E2 -22428.231} C_VEL
LIN {X 0,Y 182.513,Z 382.507,A -85,B 0,C 180,E1 -22432.458,E2 -22432.458} C_VEL
LIN {X 0,Y 186.149,Z 374.921,A -85,B 0,C 180,E1 -22436.335,E2 -22436.335} C_VEL
LIN {X 0,Y 190.35,Z 365.883,A -85,B 0,C 180,E1 -22439.897,E2 -22439.897} C_VEL
LIN {X 0,Y 194.572,Z 356.406,A -85,B 0,C 180,E1 -22442.807,E2 -22442.807} C_VEL
LIN {X 0,Y 198.665,Z 346.45,A -85,B 0,C 180,E1 -22445.246,E2 -22445.246} C_VEL
LIN {X 0,Y 199.839,Z 342.963,A -85,B 0,C 180,E1 -22446.014,E2 -22446.014} C_VEL
LIN {X 0,Y 200.295,Z 332.432,A -85,B 0,C 180,E1 -22448.654,E2 -22448.654} C_VEL
LIN {X 0,Y 199.942,Z 322.819,A -85,B 0,C 180,E1 -22450.913,E2 -22450.913} C_VEL
LIN {X 0,Y 198.698,Z 312.575,A -85,B 0,C 180,E1 -22453.267,E2 -22453.267} C_VEL
LIN {X 0,Y 196.594,Z 303.069,A -85,B 0,C 180,E1 -22455.473,E2 -22455.473} C_VEL
LIN {X 0,Y 193.446,Z 294.249,A -85,B 0,C 180,E1 -22457.77,E2 -22457.77} C_VEL
LIN {X 0,Y 190.145,Z 287.355,A -85,B 0,C 180,E1 -22459.796,E2 -22459.796} C_VEL
LIN {X 0,Y 188.431,Z 283.969,A -85,B 0,C 180,E1 -22460.811,E2 -22460.811} C_VEL
LIN {X 0,Y 186.272,Z 279.799,A -85,B 0,C 180,E1 -22462.115,E2 -22462.115} C_VEL
LIN {X 0,Y 183.68,Z 275.93,A -85,B 0,C 180,E1 -22463.547,E2 -22463.547} C_VEL
LIN {X 0,Y 182.668,Z 273.785,A -85,B 0,C 180,E1 -22464.195,E2 -22464.195} C_VEL
LIN {X 0,Y 180.356,Z 271.14,A -85,B 0,C 180,E1 -22465.451,E2 -22465.451} C_VEL
LIN {X 0,Y 179.149,Z 267.983,A -85,B 0,C 180,E1 -22466.315,E2 -22466.315} C_VEL
LIN {X 0,Y 178.883,Z 266.416,A -85,B 0,C 180,E1 -22469.808,E2 -22469.808} C_VEL
LIN {X 0,Y 178.602,Z 264.441,A -85,B 0,C 180,E1 -22474.83,E2 -22474.83} C_VEL
LIN {X 0,Y 178.493,Z 263.877,A -85,B 0,C 180,E1 -22476.813,E2 -22476.813} C_VEL
LIN {X 0,Y 178.615,Z 263.857,A -85,B 0,C 180,E1 -22481.653,E2 -22481.653} C_VEL
LIN {X 0,Y 178.648,Z 263.851,A -85,B 0,C 180,E1 -22486.347,E2 -22486.347} C_VEL
LIN {X 0,Y 178.907,Z 263.823,A -85,B 0,C 180,E1 -22490.96,E2 -22490.96} C_VEL
LIN {X 0,Y 179.15,Z 263.794,A -85,B 0,C 180,E1 -22497.752,E2 -22497.752} C_VEL
LIN {X 0,Y 179.365,Z 263.767,A -85,B 0,C 180,E1 -22500,E2 -22500} C_VEL
LIN {X 0,Y 178.865,Z 263.828,A -85,B 0,C 180,E1 -22504.507,E2 -22504.507} C_VEL
LIN {X 0,Y 178.913,Z 263.822,A -85,B 0,C 180,E1 -22509.04,E2 -22509.04} C_VEL
LIN {X 0,Y 178.66,Z 263.853,A -85,B 0,C 180,E1 -22513.652,E2 -22513.652} C_VEL
LIN {X 0,Y 178.622,Z 263.861,A -85,B 0,C 180,E1 -22519.215,E2 -22519.215} C_VEL
LIN {X 0,Y 178.521,Z 263.873,A -85,B 0,C 180,E1 -22525.114,E2 -22525.114} C_VEL
LIN {X 0,Y 178.522,Z 263.872,A -85,B 0,C 180,E1 -22529.993,E2 -22529.993} C_VEL
LIN {X 0,Y 178.594,Z 264.448,A -85,B 0,C 180,E1 -22533.504,E2 -22533.504} C_VEL
LIN {X 0,Y 179.696,Z 267.301,A -85,B 0,C 180,E1 -22534.289,E2 -22534.289} C_VEL
LIN {X 0,Y 182.016,Z 269.891,A -85,B 0,C 180,E1 -22535.58,E2 -22535.58} C_VEL
LIN {X 0,Y 184.594,Z 274.357,A -85,B 0,C 180,E1 -22537.14,E2 -22537.14} C_VEL
LIN {X 0,Y 185.868,Z 276.035,A -85,B 0,C 180,E1 -22537.833,E2 -22537.833} C_VEL
LIN {X 0,Y 188.209,Z 280.068,A -85,B 0,C 180,E1 -22539.222,E2 -22539.222} C_VEL
LIN {X 0,Y 192.382,Z 287.944,A -85,B 0,C 180,E1 -22541.726,E2 -22541.726} C_VEL
LIN {X 0,Y 196.038,Z 296.542,A -85,B 0,C 180,E1 -22544.192,E2 -22544.192} C_VEL
LIN {X 0,Y 198.551,Z 304.531,A -85,B 0,C 180,E1 -22546.284,E2 -22546.284} C_VEL
LIN {X 0,Y 200.598,Z 315.074,A -85,B 0,C 180,E1 -22548.872,E2 -22548.872} C_VEL
LIN {X 0,Y 201.692,Z 325.529,A -85,B 0,C 180,E1 -22551.475,E2 -22551.475} C_VEL
LIN {X 0,Y 201.799,Z 334.097,A -85,B 0,C 180,E1 -22553.697,E2 -22553.697} C_VEL
LIN {X 0,Y 197.863,Z 344.581,A -85,B 0,C 180,E1 -22555.984,E2 -22555.984} C_VEL
LIN {X 0,Y 193.491,Z 354.992,A -85,B 0,C 180,E1 -22558.829,E2 -22558.829} C_VEL
LIN {X 0,Y 189.487,Z 363.578,A -85,B 0,C 180,E1 -22561.778,E2 -22561.778} C_VEL
LIN {X 0,Y 185.361,Z 372.056,A -85,B 0,C 180,E1 -22565.501,E2 -22565.501} C_VEL
LIN {X 0,Y 182.899,Z 377.527,A -85,B 0,C 180,E1 -22568.59,E2 -22568.59} C_VEL
LIN {X 0,Y 180.438,Z 382.236,A -85,B 0,C 180,E1 -22571.845,E2 -22571.845} C_VEL
LIN {X 0,Y 178.235,Z 387.107,A -85,B 0,C 180,E1 -22576.315,E2 -22576.315} C_VEL
LIN {X 0,Y 176.806,Z 390.492,A -85,B 0,C 180,E1 -22580.851,E2 -22580.851} C_VEL
LIN {X 0,Y 176.151,Z 392.497,A -85,B 0,C 180,E1 -22585.423,E2 -22585.423} C_VEL
LIN {X 0,Y 176.023,Z 393.177,A -85,B 0,C 180,E1 -22590,E2 -22590} C_VEL
LIN {X 0,Y 176.151,Z 392.546,A -85,B 0,C 180,E1 -22594.577,E2 -22594.577} C_VEL
LIN {X 0,Y 176.805,Z 390.586,A -85,B 0,C 180,E1 -22599.149,E2 -22599.149} C_VEL
LIN {X 0,Y 178.208,Z 387.247,A -85,B 0,C 180,E1 -22603.688,E2 -22603.688} C_VEL
LIN {X 0,Y 180.399,Z 382.429,A -85,B 0,C 180,E1 -22608.16,E2 -22608.16} C_VEL
LIN {X 0,Y 182.831,Z 377.772,A -85,B 0,C 180,E1 -22611.419,E2 -22611.419} C_VEL
LIN {X 0,Y 185.958,Z 371.005,A -85,B 0,C 180,E1 -22615.162,E2 -22615.162} C_VEL
LIN {X 0,Y 189.404,Z 363.938,A -85,B 0,C 180,E1 -22618.236,E2 -22618.236} C_VEL
LIN {X 0,Y 193.392,Z 355.423,A -85,B 0,C 180,E1 -22621.189,E2 -22621.189} C_VEL
LIN {X 0,Y 197.731,Z 345.1,A -85,B 0,C 180,E1 -22624.043,E2 -22624.043} C_VEL
LIN {X 0,Y 201.765,Z 334.719,A -85,B 0,C 180,E1 -22626.31,E2 -22626.31} C_VEL
LIN {X 0,Y 201.842,Z 327.479,A -85,B 0,C 180,E1 -22628.173,E2 -22628.173} C_VEL
LIN {X 0,Y 200.922,Z 316.81,A -85,B 0,C 180,E1 -22630.852,E2 -22630.852} C_VEL
LIN {X 0,Y 199.275,Z 307.225,A -85,B 0,C 180,E1 -22633.217,E2 -22633.217} C_VEL
LIN {X 0,Y 197.017,Z 299.126,A -85,B 0,C 180,E1 -22635.28,E2 -22635.28} C_VEL
LIN {X 0,Y 194.228,Z 291.922,A -85,B 0,C 180,E1 -22637.277,E2 -22637.277} C_VEL
LIN {X 0,Y 190.303,Z 283.931,A -85,B 0,C 180,E1 -22639.732,E2 -22639.732} C_VEL
LIN {X 0,Y 187.739,Z 279.353,A -85,B 0,C 180,E1 -22641.251,E2 -22641.251} C_VEL
LIN {X 0,Y 185.199,Z 274.992,A -85,B 0,C 180,E1 -22642.768,E2 -22642.768} C_VEL
LIN {X 0,Y 183.032,Z 271.884,A -85,B 0,C 180,E1 -22643.995,E2 -22643.995} C_VEL
LIN {X 0,Y 182.07,Z 269.96,A -85,B 0,C 180,E1 -22644.619,E2 -22644.619} C_VEL
LIN {X 0,Y 179.767,Z 267.428,A -85,B 0,C 180,E1 -22645.904,E2 -22645.904} C_VEL
LIN {X 0,Y 178.593,Z 264.455,A -85,B 0,C 180,E1 -22646.738,E2 -22646.738} C_VEL
LIN {X 0,Y 178.525,Z 263.873,A -85,B 0,C 180,E1 -22650.006,E2 -22650.006} C_VEL
LIN {X 0,Y 178.522,Z 263.865,A -85,B 0,C 180,E1 -22654.886,E2 -22654.886} C_VEL
LIN {X 0,Y 178.624,Z 263.861,A -85,B 0,C 180,E1 -22660.786,E2 -22660.786} C_VEL
LIN {X 0,Y 178.66,Z 263.854,A -85,B 0,C 180,E1 -22666.348,E2 -22666.348} C_VEL
LIN {X 0,Y 178.913,Z 263.824,A -85,B 0,C 180,E1 -22670.96,E2 -22670.96} C_VEL
LIN {X 0,Y 179.152,Z 263.792,A -85,B 0,C 180,E1 -22677.752,E2 -22677.752} C_VEL
LIN {X 0,Y 179.354,Z 263.767,A -85,B 0,C 180,E1 -22680,E2 -22680} C_VEL
LIN {X 0,Y 178.861,Z 263.829,A -85,B 0,C 180,E1 -22684.507,E2 -22684.507} C_VEL
LIN {X 0,Y 178.908,Z 263.826,A -85,B 0,C 180,E1 -22689.04,E2 -22689.04} C_VEL
LIN {X 0,Y 178.65,Z 263.859,A -85,B 0,C 180,E1 -22693.653,E2 -22693.653} C_VEL
LIN {X 0,Y 178.622,Z 263.859,A -85,B 0,C 180,E1 -22699.213,E2 -22699.213} C_VEL
LIN {X 0,Y 178.495,Z 263.875,A -85,B 0,C 180,E1 -22703.187,E2 -22703.187} C_VEL
LIN {X 0,Y 178.727,Z 265.656,A -85,B 0,C 180,E1 -22708.156,E2 -22708.156} C_VEL
LIN {X 0,Y 179.135,Z 267.966,A -85,B 0,C 180,E1 -22713.503,E2 -22713.503} C_VEL
LIN {X 0,Y 180.468,Z 271.314,A -85,B 0,C 180,E1 -22714.471,E2 -22714.471} C_VEL
LIN {X 0,Y 183.092,Z 274.398,A -85,B 0,C 180,E1 -22715.915,E2 -22715.915} C_VEL
LIN {X 0,Y 184.87,Z 277.967,A -85,B 0,C 180,E1 -22717.017,E2 -22717.017} C_VEL
LIN {X 0,Y 186.449,Z 280.142,A -85,B 0,C 180,E1 -22717.867,E2 -22717.867} C_VEL
LIN {X 0,Y 188.589,Z 284.154,A -85,B 0,C 180,E1 -22719.15,E2 -22719.15} C_VEL
LIN {X 0,Y 191.781,Z 290.614,A -85,B 0,C 180,E1 -22721.088,E2 -22721.088} C_VEL
LIN {X 0,Y 195.044,Z 298.192,A -85,B 0,C 180,E1 -22723.206,E2 -22723.206} C_VEL
LIN {X 0,Y 197.636,Z 306.802,A -85,B 0,C 180,E1 -22725.333,E2 -22725.333} C_VEL
LIN {X 0,Y 199.624,Z 318.452,A -85,B 0,C 180,E1 -22728.016,E2 -22728.016} C_VEL
LIN {X 0,Y 200.385,Z 329.082,A -85,B 0,C 180,E1 -22730.497,E2 -22730.497} C_VEL
LIN {X 0,Y 200.068,Z 340.68,A -85,B 0,C 180,E1 -22733.332,E2 -22733.332} C_VEL
LIN {X 0,Y 199.707,Z 343.895,A -85,B 0,C 180,E1 -22734.153,E2 -22734.153} C_VEL
LIN {X 0,Y 195.351,Z 354.832,A -85,B 0,C 180,E1 -22736.726,E2 -22736.726} C_VEL
LIN {X 0,Y 190.994,Z 364.568,A -85,B 0,C 180,E1 -22739.605,E2 -22739.605} C_VEL
LIN {X 0,Y 187.279,Z 372.65,A -85,B 0,C 180,E1 -22742.632,E2 -22742.632} C_VEL
LIN {X 0,Y 183.644,Z 380.401,A -85,B 0,C 180,E1 -22746.307,E2 -22746.307} C_VEL
LIN {X 0,Y 181.148,Z 385.813,A -85,B 0,C 180,E1 -22749.563,E2 -22749.563} C_VEL
LIN {X 0,Y 178.481,Z 391.51,A -85,B 0,C 180,E1 -22754,E2 -22754} C_VEL
LIN {X 0,Y 176.863,Z 395.648,A -85,B 0,C 180,E1 -22758.54,E2 -22758.54} C_VEL
LIN {X 0,Y 176.079,Z 398.354,A -85,B 0,C 180,E1 -22763.123,E2 -22763.123} C_VEL
LIN {X 0,Y 175.887,Z 399.693,A -85,B 0,C 180,E1 -22767.71,E2 -22767.71} C_VEL
LIN {X 0,Y 175.999,Z 399.856,A -85,B 0,C 180,E1 -22769.965,E2 -22769.965} C_VEL
LIN {X 0,Y 175.455,Z 399.833,A -85,B 0,C 180,E1 -22771.873,E2 -22771.873} C_VEL
LIN {X 0,Y 173.895,Z 399.518,A -85,B 0,C 180,E1 -22773.75,E2 -22773.75} C_VEL
LIN {X 0,Y 170.238,Z 398.1,A -85,B 0,C 180,E1 -22777.54,E2 -22777.54} C_VEL
LIN {X 0,Y 169.397,Z 397.029,A -85,B 0,C 180,E1 -22779.509,E2 -22779.509} C_VEL
LIN {X 0,Y 169.429,Z 396.607,A -85,B 0,C 180,E1 -22780.17,E2 -22780.17} C_VEL
LIN {X 0,Y 170.574,Z 393.57,A -85,B 0,C 180,E1 -22784.312,E2 -22784.312} C_VEL
LIN {X 0,Y 172.921,Z 388.646,A -85,B 0,C 180,E1 -22788.974,E2 -22788.974} C_VEL
LIN {X 0,Y 175.696,Z 382.819,A -85,B 0,C 180,E1 -22793.071,E2 -22793.071} C_VEL
LIN {X 0,Y 179.19,Z 375.904,A -85,B 0,C 180,E1 -22796.81,E2 -22796.81} C_VEL
LIN {X 0,Y 183.522,Z 367.138,A -85,B 0,C 180,E1 -22800.491,E2 -22800.491} C_VEL
LIN {X 0,Y 187.854,Z 357.97,A -85,B 0,C 180,E1 -22803.492,E2 -22803.492} C_VEL
LIN {X 0,Y 192.459,Z 347.425,A -85,B 0,C 180,E1 -22806.216,E2 -22806.216} C_VEL
LIN {X 0,Y 193.622,Z 343.988,A -85,B 0,C 180,E1 -22807.009,E2 -22807.009} C_VEL
LIN {X 0,Y 194.244,Z 333.698,A -85,B 0,C 180,E1 -22809.729,E2 -22809.729} C_VEL
LIN {X 0,Y 194.044,Z 324.227,A -85,B 0,C 180,E1 -22812.097,E2 -22812.097} C_VEL
LIN {X 0,Y 192.821,Z 313.374,A -85,B 0,C 180,E1 -22814.741,E2 -22814.741} C_VEL
LIN {X 0,Y 190.958,Z 305.167,A -85,B 0,C 180,E1 -22816.836,E2 -22816.836} C_VEL
LIN {X 0,Y 188.778,Z 298.728,A -85,B 0,C 180,E1 -22818.638,E2 -22818.638} C_VEL
LIN {X 0,Y 184.637,Z 289.5,A -85,B 0,C 180,E1 -22821.53,E2 -22821.53} C_VEL
LIN {X 0,Y 181.878,Z 284.31,A -85,B 0,C 180,E1 -22823.346,E2 -22823.346} C_VEL
LIN {X 0,Y 179.805,Z 280.5,A -85,B 0,C 180,E1 -22824.733,E2 -22824.733} C_VEL
LIN {X 0,Y 178.889,Z 279.113,A -85,B 0,C 180,E1 -22825.315,E2 -22825.315} C_VEL
LIN {X 0,Y 176.627,Z 275.73,A -85,B 0,C 180,E1 -22826.762,E2 -22826.762} C_VEL
LIN {X 0,Y 175.862,Z 273.929,A -85,B 0,C 180,E1 -22827.349,E2 -22827.349} C_VEL
LIN {X 0,Y 173.307,Z 271.187,A -85,B 0,C 180,E1 -22828.966,E2 -22828.966} C_VEL
LIN {X 0,Y 171.961,Z 267.985,A -85,B 0,C 180,E1 -22830.023,E2 -22830.023} C_VEL
LIN {X 0,Y 171.847,Z 267.544,A -85,B 0,C 180,E1 -22830.61,E2 -22830.61} C_VEL
LIN {X 0,Y 171.576,Z 265.618,A -85,B 0,C 180,E1 -22835.82,E2 -22835.82} C_VEL
LIN {X 0,Y 171.445,Z 264.792,A -85,B 0,C 180,E1 -22838.35,E2 -22838.35} C_VEL
LIN {X 0,Y 171.547,Z 264.743,A -85,B 0,C 180,E1 -22840.868,E2 -22840.868} C_VEL
LIN {X 0,Y 171.562,Z 264.732,A -85,B 0,C 180,E1 -22845.772,E2 -22845.772} C_VEL
LIN {X 0,Y 171.845,Z 264.699,A -85,B 0,C 180,E1 -22850.585,E2 -22850.585} C_VEL
LIN {X 0,Y 171.808,Z 264.708,A -85,B 0,C 180,E1 -22855.307,E2 -22855.307} C_VEL
LIN {X 0,Y 172.328,Z 264.643,A -85,B 0,C 180,E1 -22860,E2 -22860} C_VEL
LIN {X 0,Y 171.813,Z 264.707,A -85,B 0,C 180,E1 -22864.693,E2 -22864.693} C_VEL
LIN {X 0,Y 171.849,Z 264.702,A -85,B 0,C 180,E1 -22869.415,E2 -22869.415} C_VEL
LIN {X 0,Y 171.578,Z 264.736,A -85,B 0,C 180,E1 -22874.227,E2 -22874.227} C_VEL
LIN {X 0,Y 171.542,Z 264.742,A -85,B 0,C 180,E1 -22879.558,E2 -22879.558} C_VEL
LIN {X 0,Y 171.459,Z 264.751,A -85,B 0,C 180,E1 -22885.609,E2 -22885.609} C_VEL
LIN {X 0,Y 171.472,Z 264.819,A -85,B 0,C 180,E1 -22889.745,E2 -22889.745} C_VEL
LIN {X 0,Y 172.348,Z 267.436,A -85,B 0,C 180,E1 -22890.507,E2 -22890.507} C_VEL
LIN {X 0,Y 174.257,Z 269.786,A -85,B 0,C 180,E1 -22891.792,E2 -22891.792} C_VEL
LIN {X 0,Y 175.678,Z 271.079,A -85,B 0,C 180,E1 -22892.69,E2 -22892.69} C_VEL
LIN {X 0,Y 177.657,Z 274.585,A -85,B 0,C 180,E1 -22894.074,E2 -22894.074} C_VEL
LIN {X 0,Y 179.167,Z 276.471,A -85,B 0,C 180,E1 -22895.009,E2 -22895.009} C_VEL
LIN {X 0,Y 181.243,Z 280.161,A -85,B 0,C 180,E1 -22896.422,E2 -22896.422} C_VEL
LIN {X 0,Y 182.414,Z 282.09,A -85,B 0,C 180,E1 -22897.167,E2 -22897.167} C_VEL
LIN {X 0,Y 185.571,Z 287.985,A -85,B 0,C 180,E1 -22899.285,E2 -22899.285} C_VEL
LIN {X 0,Y 189.312,Z 296.026,A -85,B 0,C 180,E1 -22901.931,E2 -22901.931} C_VEL
LIN {X 0,Y 192.239,Z 304.349,A -85,B 0,C 180,E1 -22904.389,E2 -22904.389} C_VEL
LIN {X 0,Y 194.179,Z 313.077,A -85,B 0,C 180,E1 -22906.714,E2 -22906.714} C_VEL
LIN {X 0,Y 195.403,Z 323.643,A -85,B 0,C 180,E1 -22909.486,E2 -22909.486} C_VEL
LIN {X 0,Y 195.68,Z 332.244,A -85,B 0,C 180,E1 -22911.806,E2 -22911.806} C_VEL
LIN {X 0,Y 195.468,Z 336.215,A -85,B 0,C 180,E1 -22912.877,E2 -22912.877} C_VEL
LIN {X 0,Y 191.215,Z 346.631,A -85,B 0,C 180,E1 -22915.271,E2 -22915.271} C_VEL
LIN {X 0,Y 186.707,Z 356.663,A -85,B 0,C 180,E1 -22918.198,E2 -22918.198} C_VEL
LIN {X 0,Y 182.607,Z 364.991,A -85,B 0,C 180,E1 -22921.244,E2 -22921.244} C_VEL
LIN {X 0,Y 178.71,Z 372.566,A -85,B 0,C 180,E1 -22924.757,E2 -22924.757} C_VEL
LIN {X 0,Y 175.391,Z 379.333,A -85,B 0,C 180,E1 -22928.861,E2 -22928.861} C_VEL
LIN {X 0,Y 172.343,Z 385.002,A -85,B 0,C 180,E1 -22933.414,E2 -22933.414} C_VEL
LIN {X 0,Y 170.449,Z 389.113,A -85,B 0,C 180,E1 -22938.103,E2 -22938.103} C_VEL
LIN {X 0,Y 169.349,Z 391.798,A -85,B 0,C 180,E1 -22942.848,E2 -22942.848} C_VEL
LIN {X 0,Y 168.948,Z 393.136,A -85,B 0,C 180,E1 -22947.616,E2 -22947.616} C_VEL
LIN {X 0,Y 168.937,Z 393.311,A -85,B 0,C 180,E1 -22950,E2 -22950} C_VEL
LIN {X 0,Y 169.07,Z 392.681,A -85,B 0,C 180,E1 -22954.769,E2 -22954.769} C_VEL
LIN {X 0,Y 169.787,Z 390.72,A -85,B 0,C 180,E1 -22959.531,E2 -22959.531} C_VEL
LIN {X 0,Y 171.275,Z 387.382,A -85,B 0,C 180,E1 -22964.253,E2 -22964.253} C_VEL
LIN {X 0,Y 173.664,Z 382.563,A -85,B 0,C 180,E1 -22968.89,E2 -22968.89} C_VEL
LIN {X 0,Y 176.199,Z 377.906,A -85,B 0,C 180,E1 -22972.267,E2 -22972.267} C_VEL
LIN {X 0,Y 179.539,Z 371.139,A -85,B 0,C 180,E1 -22976.128,E2 -22976.128} C_VEL
LIN {X 0,Y 183.178,Z 364.071,A -85,B 0,C 180,E1 -22979.287,E2 -22979.287} C_VEL
LIN {X 0,Y 187.332,Z 355.556,A -85,B 0,C 180,E1 -22982.318,E2 -22982.318} C_VEL
LIN {X 0,Y 191.894,Z 345.232,A -85,B 0,C 180,E1 -22985.228,E2 -22985.228} C_VEL
LIN {X 0,Y 195.472,Z 336.528,A -85,B 0,C 180,E1 -22987.199,E2 -22987.199} C_VEL
LIN {X 0,Y 195.8,Z 332.56,A -85,B 0,C 180,E1 -22988.249,E2 -22988.249} C_VEL
LIN {X 0,Y 195.56,Z 323.984,A -85,B 0,C 180,E1 -22990.568,E2 -22990.568} C_VEL
LIN {X 0,Y 194.554,Z 314.765,A -85,B 0,C 180,E1 -22992.989,E2 -22992.989} C_VEL
LIN {X 0,Y 192.636,Z 305.487,A -85,B 0,C 180,E1 -22995.464,E2 -22995.464} C_VEL
LIN {X 0,Y 190.083,Z 297.851,A -85,B 0,C 180,E1 -22997.687,E2 -22997.687} C_VEL
LIN {X 0,Y 186.68,Z 289.917,A -85,B 0,C 180,E1 -23000.208,E2 -23000.208} C_VEL
LIN {X 0,Y 183.355,Z 283.86,A -85,B 0,C 180,E1 -23002.407,E2 -23002.407} C_VEL
LIN {X 0,Y 181.42,Z 280.349,A -85,B 0,C 180,E1 -23003.705,E2 -23003.705} C_VEL
LIN {X 0,Y 179.216,Z 276.503,A -85,B 0,C 180,E1 -23005.2,E2 -23005.2} C_VEL
LIN {X 0,Y 176.277,Z 272.429,A -85,B 0,C 180,E1 -23007.097,E2 -23007.097} C_VEL
LIN {X 0,Y 175.411,Z 270.519,A -85,B 0,C 180,E1 -23007.766,E2 -23007.766} C_VEL
LIN {X 0,Y 172.849,Z 268.178,A -85,B 0,C 180,E1 -23009.405,E2 -23009.405} C_VEL
LIN {X 0,Y 171.644,Z 265.667,A -85,B 0,C 180,E1 -23010.344,E2 -23010.344} C_VEL
LIN {X 0,Y 171.448,Z 264.754,A -85,B 0,C 180,E1 -23010.618,E2 -23010.618} C_VEL
LIN {X 0,Y 171.447,Z 264.748,A -85,B 0,C 180,E1 -23015.8,E2 -23015.8} C_VEL
LIN {X 0,Y 171.58,Z 264.739,A -85,B 0,C 180,E1 -23020.872,E2 -23020.872} C_VEL
LIN {X 0,Y 171.579,Z 264.738,A -85,B 0,C 180,E1 -23025.773,E2 -23025.773} C_VEL
LIN {X 0,Y 171.85,Z 264.705,A -85,B 0,C 180,E1 -23030.585,E2 -23030.585} C_VEL
LIN {X 0,Y 171.813,Z 264.707,A -85,B 0,C 180,E1 -23035.307,E2 -23035.307} C_VEL
LIN {X 0,Y 172.319,Z 264.643,A -85,B 0,C 180,E1 -23040,E2 -23040} C_VEL
LIN {X 0,Y 171.809,Z 264.707,A -85,B 0,C 180,E1 -23044.693,E2 -23044.693} C_VEL
LIN {X 0,Y 171.846,Z 264.703,A -85,B 0,C 180,E1 -23049.415,E2 -23049.415} C_VEL
LIN {X 0,Y 171.567,Z 264.739,A -85,B 0,C 180,E1 -23054.228,E2 -23054.228} C_VEL
LIN {X 0,Y 171.541,Z 264.742,A -85,B 0,C 180,E1 -23059.556,E2 -23059.556} C_VEL
LIN {X 0,Y 171.45,Z 264.861,A -85,B 0,C 180,E1 -23061.649,E2 -23061.649} C_VEL
LIN {X 0,Y 171.667,Z 266.234,A -85,B 0,C 180,E1 -23065.752,E2 -23065.752} C_VEL
LIN {X 0,Y 171.917,Z 267.84,A -85,B 0,C 180,E1 -23069.757,E2 -23069.757} C_VEL
LIN {X 0,Y 173.302,Z 271.171,A -85,B 0,C 180,E1 -23070.858,E2 -23070.858} C_VEL
LIN {X 0,Y 175.846,Z 273.917,A -85,B 0,C 180,E1 -23072.483,E2 -23072.483} C_VEL
LIN {X 0,Y 178.029,Z 278.077,A -85,B 0,C 180,E1 -23074.024,E2 -23074.024} C_VEL
LIN {X 0,Y 179.724,Z 280.297,A -85,B 0,C 180,E1 -23075.062,E2 -23075.062} C_VEL
LIN {X 0,Y 181.862,Z 284.28,A -85,B 0,C 180,E1 -23076.509,E2 -23076.509} C_VEL
LIN {X 0,Y 183.043,Z 286.5,A -85,B 0,C 180,E1 -23077.279,E2 -23077.279} C_VEL
LIN {X 0,Y 185.339,Z 290.929,A -85,B 0,C 180,E1 -23078.819,E2 -23078.819} C_VEL
LIN {X 0,Y 189.593,Z 300.736,A -85,B 0,C 180,E1 -23081.854,E2 -23081.854} C_VEL
LIN {X 0,Y 191.995,Z 308.895,A -85,B 0,C 180,E1 -23084.067,E2 -23084.067} C_VEL
LIN {X 0,Y 193.674,Z 318.881,A -85,B 0,C 180,E1 -23086.532,E2 -23086.532} C_VEL
LIN {X 0,Y 194.339,Z 329.076,A -85,B 0,C 180,E1 -23089.045,E2 -23089.045} C_VEL
LIN {X 0,Y 194.095,Z 338.599,A -85,B 0,C 180,E1 -23091.466,E2 -23091.466} C_VEL
LIN {X 0,Y 193.677,Z 344.141,A -85,B 0,C 180,E1 -23092.97,E2 -23092.97} C_VEL
LIN {X 0,Y 189.444,Z 354.7,A -85,B 0,C 180,E1 -23095.546,E2 -23095.546} C_VEL
LIN {X 0,Y 184.877,Z 364.435,A -85,B 0,C 180,E1 -23098.486,E2 -23098.486} C_VEL
LIN {X 0,Y 180.956,Z 372.516,A -85,B 0,C 180,E1 -23101.59,E2 -23101.59} C_VEL
LIN {X 0,Y 177.107,Z 380.266,A -85,B 0,C 180,E1 -23105.376,E2 -23105.376} C_VEL
LIN {X 0,Y 174.473,Z 385.679,A -85,B 0,C 180,E1 -23108.744,E2 -23108.744} C_VEL
LIN {X 0,Y 171.642,Z 391.376,A -85,B 0,C 180,E1 -23113.344,E2 -23113.344} C_VEL
LIN {X 0,Y 169.856,Z 395.513,A -85,B 0,C 180,E1 -23118.06,E2 -23118.06} C_VEL
LIN {X 0,Y 168.997,Z 398.219,A -85,B 0,C 180,E1 -23122.833,E2 -23122.833} C_VEL
LIN {X 0,Y 168.854,Z 399.058,A -85,B 0,C 180,E1 -23125.225,E2 -23125.225} C_VEL
LIN {X 0,Y 168.914,Z 399.724,A -85,B 0,C 180,E1 -23130,E2 -23130} C_VEL
LIN {X 0,Y 168.852,Z 399.037,A -85,B 0,C 180,E1 -23134.775,E2 -23134.775} C_VEL
LIN {X 0,Y 169.32,Z 397.001,A -85,B 0,C 180,E1 -23139.557,E2 -23139.557} C_VEL
LIN {X 0,Y 169.429,Z 396.607,A -85,B 0,C 180,E1 -23140.17,E2 -23140.17} C_VEL
LIN {X 0,Y 169.218,Z 395.364,A -85,B 0,C 180,E1 -23142.118,E2 -23142.118} C_VEL
LIN {X 0,Y 167.44,Z 392.859,A -85,B 0,C 180,E1 -23145.331,E2 -23145.331} C_VEL
LIN {X 0,Y 166.217,Z 390.504,A -85,B 0,C 180,E1 -23147.911,E2 -23147.911} C_VEL
LIN {X 0,Y 166.28,Z 388.442,A -85,B 0,C 180,E1 -23149.828,E2 -23149.828} C_VEL
LIN {X 0,Y 166.6,Z 387.692,A -85,B 0,C 180,E1 -23150.45,E2 -23150.45} C_VEL
LIN {X 0,Y 169.544,Z 381.944,A -85,B 0,C 180,E1 -23154.489,E2 -23154.489} C_VEL
LIN {X 0,Y 173.456,Z 374.646,A -85,B 0,C 180,E1 -23158.43,E2 -23158.43} C_VEL
LIN {X 0,Y 178.096,Z 365.607,A -85,B 0,C 180,E1 -23162.19,E2 -23162.19} C_VEL
LIN {X 0,Y 182.781,Z 356.131,A -85,B 0,C 180,E1 -23165.223,E2 -23165.223} C_VEL
LIN {X 0,Y 186.869,Z 346.956,A -85,B 0,C 180,E1 -23167.592,E2 -23167.592} C_VEL
LIN {X 0,Y 187.444,Z 345.059,A -85,B 0,C 180,E1 -23168.059,E2 -23168.059} C_VEL
LIN {X 0,Y 188.305,Z 333.546,A -85,B 0,C 180,E1 -23171.248,E2 -23171.248} C_VEL
LIN {X 0,Y 188.047,Z 323.09,A -85,B 0,C 180,E1 -23173.997,E2 -23173.997} C_VEL
LIN {X 0,Y 186.918,Z 313.896,A -85,B 0,C 180,E1 -23176.412,E2 -23176.412} C_VEL
LIN {X 0,Y 185.26,Z 306.814,A -85,B 0,C 180,E1 -23178.404,E2 -23178.404} C_VEL
LIN {X 0,Y 182.071,Z 298.188,A -85,B 0,C 180,E1 -23181.152,E2 -23181.152} C_VEL
LIN {X 0,Y 178.149,Z 289.801,A -85,B 0,C 180,E1 -23184.156,E2 -23184.156} C_VEL
LIN {X 0,Y 175.475,Z 284.834,A -85,B 0,C 180,E1 -23186.151,E2 -23186.151} C_VEL
LIN {X 0,Y 173.17,Z 280.927,A -85,B 0,C 180,E1 -23187.868,E2 -23187.868} C_VEL
LIN {X 0,Y 172.479,Z 279.625,A -85,B 0,C 180,E1 -23188.425,E2 -23188.425} C_VEL
LIN {X 0,Y 170.091,Z 276.452,A -85,B 0,C 180,E1 -23190.162,E2 -23190.162} C_VEL
LIN {X 0,Y 168.873,Z 273.82,A -85,B 0,C 180,E1 -23191.237,E2 -23191.237} C_VEL
LIN {X 0,Y 166.241,Z 271.117,A -85,B 0,C 180,E1 -23193.262,E2 -23193.262} C_VEL
LIN {X 0,Y 164.818,Z 268.015,A -85,B 0,C 180,E1 -23194.616,E2 -23194.616} C_VEL
LIN {X 0,Y 164.696,Z 267.442,A -85,B 0,C 180,E1 -23194.909,E2 -23194.909} C_VEL
LIN {X 0,Y 164.482,Z 265.835,A -85,B 0,C 180,E1 -23200.054,E2 -23200.054} C_VEL
LIN {X 0,Y 164.49,Z 265.614,A -85,B 0,C 180,E1 -23205.146,E2 -23205.146} C_VEL
LIN {X 0,Y 164.766,Z 265.578,A -85,B 0,C 180,E1 -23210.176,E2 -23210.176} C_VEL
LIN {X 0,Y 164.825,Z 265.577,A -85,B 0,C 180,E1 -23212.651,E2 -23212.651} C_VEL
LIN {X 0,Y 165.045,Z 265.55,A -85,B 0,C 180,E1 -23217.56,E2 -23217.56} C_VEL
LIN {X 0,Y 165.291,Z 265.52,A -85,B 0,C 180,E1 -23220,E2 -23220} C_VEL
LIN {X 0,Y 164.762,Z 265.585,A -85,B 0,C 180,E1 -23224.894,E2 -23224.894} C_VEL
LIN {X 0,Y 164.832,Z 265.577,A -85,B 0,C 180,E1 -23227.349,E2 -23227.349} C_VEL
LIN {X 0,Y 164.704,Z 265.592,A -85,B 0,C 180,E1 -23231.062,E2 -23231.062} C_VEL
LIN {X 0,Y 164.484,Z 265.621,A -85,B 0,C 180,E1 -23237.403,E2 -23237.403} C_VEL
LIN {X 0,Y 164.474,Z 265.621,A -85,B 0,C 180,E1 -23239.989,E2 -23239.989} C_VEL
LIN {X 0,Y 164.425,Z 265.628,A -85,B 0,C 180,E1 -23245.136,E2 -23245.136} C_VEL
LIN {X 0,Y 165.248,Z 268.222,A -85,B 0,C 180,E1 -23246.08,E2 -23246.08} C_VEL
LIN {X 0,Y 167.033,Z 270.337,A -85,B 0,C 180,E1 -23247.57,E2 -23247.57} C_VEL
LIN {X 0,Y 168.815,Z 271.655,A -85,B 0,C 180,E1 -23248.898,E2 -23248.898} C_VEL
LIN {X 0,Y 170.623,Z 275.004,A -85,B 0,C 180,E1 -23250.423,E2 -23250.423} C_VEL
LIN {X 0,Y 172.686,Z 277.222,A -85,B 0,C 180,E1 -23251.886,E2 -23251.886} C_VEL
LIN {X 0,Y 174.832,Z 280.932,A -85,B 0,C 180,E1 -23253.548,E2 -23253.548} C_VEL
LIN {X 0,Y 175.776,Z 282.331,A -85,B 0,C 180,E1 -23254.212,E2 -23254.212} C_VEL
LIN {X 0,Y 179.115,Z 288.616,A -85,B 0,C 180,E1 -23256.754,E2 -23256.754} C_VEL
LIN {X 0,Y 183.17,Z 296.927,A -85,B 0,C 180,E1 -23259.881,E2 -23259.881} C_VEL
LIN {X 0,Y 186.352,Z 305.731,A -85,B 0,C 180,E1 -23262.754,E2 -23262.754} C_VEL
LIN {X 0,Y 187.986,Z 312.464,A -85,B 0,C 180,E1 -23264.738,E2 -23264.738} C_VEL
LIN {X 0,Y 189.234,Z 321.938,A -85,B 0,C 180,E1 -23267.393,E2 -23267.393} C_VEL
LIN {X 0,Y 189.659,Z 332.468,A -85,B 0,C 180,E1 -23270.382,E2 -23270.382} C_VEL
LIN {X 0,Y 189.398,Z 337.479,A -85,B 0,C 180,E1 -23271.831,E2 -23271.831} C_VEL
LIN {X 0,Y 184.587,Z 348.546,A -85,B 0,C 180,E1 -23274.505,E2 -23274.505} C_VEL
LIN {X 0,Y 179.955,Z 358.28,A -85,B 0,C 180,E1 -23277.521,E2 -23277.521} C_VEL
LIN {X 0,Y 175.728,Z 366.355,A -85,B 0,C 180,E1 -23280.665,E2 -23280.665} C_VEL
LIN {X 0,Y 171.585,Z 374.075,A -85,B 0,C 180,E1 -23284.524,E2 -23284.524} C_VEL
LIN {X 0,Y 168.776,Z 379.469,A -85,B 0,C 180,E1 -23287.99,E2 -23287.99} C_VEL
LIN {X 0,Y 165.516,Z 385.139,A -85,B 0,C 180,E1 -23292.709,E2 -23292.709} C_VEL
LIN {X 0,Y 163.485,Z 389.249,A -85,B 0,C 180,E1 -23297.588,E2 -23297.588} C_VEL
LIN {X 0,Y 162.296,Z 391.933,A -85,B 0,C 180,E1 -23302.536,E2 -23302.536} C_VEL
LIN {X 0,Y 161.866,Z 393.27,A -85,B 0,C 180,E1 -23307.512,E2 -23307.512} C_VEL
LIN {X 0,Y 161.838,Z 393.446,A -85,B 0,C 180,E1 -23310,E2 -23310} C_VEL
LIN {X 0,Y 162.005,Z 392.815,A -85,B 0,C 180,E1 -23314.978,E2 -23314.978} C_VEL
LIN {X 0,Y 162.77,Z 390.855,A -85,B 0,C 180,E1 -23319.946,E2 -23319.946} C_VEL
LIN {X 0,Y 164.371,Z 387.516,A -85,B 0,C 180,E1 -23324.865,E2 -23324.865} C_VEL
LIN {X 0,Y 166.961,Z 382.697,A -85,B 0,C 180,E1 -23329.679,E2 -23329.679} C_VEL
LIN {X 0,Y 169.591,Z 378.04,A -85,B 0,C 180,E1 -23333.184,E2 -23333.184} C_VEL
LIN {X 0,Y 173.159,Z 371.272,A -85,B 0,C 180,E1 -23337.168,E2 -23337.168} C_VEL
LIN {X 0,Y 177.728,Z 362.855,A -85,B 0,C 180,E1 -23340.935,E2 -23340.935} C_VEL
LIN {X 0,Y 182.135,Z 354.068,A -85,B 0,C 180,E1 -23344.022,E2 -23344.022} C_VEL
LIN {X 0,Y 186.142,Z 345.363,A -85,B 0,C 180,E1 -23346.489,E2 -23346.489} C_VEL
LIN {X 0,Y 189.388,Z 337.821,A -85,B 0,C 180,E1 -23348.239,E2 -23348.239} C_VEL
LIN {X 0,Y 189.772,Z 331.998,A -85,B 0,C 180,E1 -23349.908,E2 -23349.908} C_VEL
LIN {X 0,Y 189.375,Z 322.576,A -85,B 0,C 180,E1 -23352.588,E2 -23352.588} C_VEL
LIN {X 0,Y 188.227,Z 313.336,A -85,B 0,C 180,E1 -23355.188,E2 -23355.188} C_VEL
LIN {X 0,Y 186.535,Z 306.161,A -85,B 0,C 180,E1 -23357.298,E2 -23357.298} C_VEL
LIN {X 0,Y 183.662,Z 298.026,A -85,B 0,C 180,E1 -23359.936,E2 -23359.936} C_VEL
LIN {X 0,Y 179.365,Z 288.988,A -85,B 0,C 180,E1 -23363.306,E2 -23363.306} C_VEL
LIN {X 0,Y 177.491,Z 285.507,A -85,B 0,C 180,E1 -23364.7,E2 -23364.7} C_VEL
LIN {X 0,Y 175.243,Z 281.376,A -85,B 0,C 180,E1 -23366.432,E2 -23366.432} C_VEL
LIN {X 0,Y 172.978,Z 277.873,A -85,B 0,C 180,E1 -23368.117,E2 -23368.117} C_VEL
LIN {X 0,Y 172.253,Z 276.499,A -85,B 0,C 180,E1 -23368.722,E2 -23368.722} C_VEL
LIN {X 0,Y 169.741,Z 273.646,A -85,B 0,C 180,E1 -23370.549,E2 -23370.549} C_VEL
LIN {X 0,Y 168.659,Z 271.283,A -85,B 0,C 180,E1 -23371.536,E2 -23371.536} C_VEL
LIN {X 0,Y 166.088,Z 269.422,A -85,B 0,C 180,E1 -23373.499,E2 -23373.499} C_VEL
LIN {X 0,Y 164.739,Z 267.038,A -85,B 0,C 180,E1 -23374.747,E2 -23374.747} C_VEL
LIN {X 0,Y 164.398,Z 265.624,A -85,B 0,C 180,E1 -23375.198,E2 -23375.198} C_VEL
LIN {X 0,Y 164.487,Z 265.619,A -85,B 0,C 180,E1 -23380.051,E2 -23380.051} C_VEL
LIN {X 0,Y 164.526,Z 265.616,A -85,B 0,C 180,E1 -23385.149,E2 -23385.149} C_VEL
LIN {X 0,Y 164.77,Z 265.585,A -85,B 0,C 180,E1 -23390.176,E2 -23390.176} C_VEL
LIN {X 0,Y 164.831,Z 265.577,A -85,B 0,C 180,E1 -23392.651,E2 -23392.651} C_VEL
LIN {X 0,Y 165.047,Z 265.548,A -85,B 0,C 180,E1 -23397.559,E2 -23397.559} C_VEL
LIN {X 0,Y 165.283,Z 265.519,A -85,B 0,C 180,E1 -23400,E2 -23400} C_VEL
LIN {X 0,Y 164.758,Z 265.585,A -85,B 0,C 180,E1 -23404.894,E2 -23404.894} C_VEL
LIN {X 0,Y 164.827,Z 265.576,A -85,B 0,C 180,E1 -23407.349,E2 -23407.349} C_VEL
LIN {X 0,Y 164.704,Z 265.596,A -85,B 0,C 180,E1 -23411.059,E2 -23411.059} C_VEL
LIN {X 0,Y 164.478,Z 265.622,A -85,B 0,C 180,E1 -23417.404,E2 -23417.404} C_VEL
LIN {X 0,Y 164.522,Z 265.911,A -85,B 0,C 180,E1 -23419.983,E2 -23419.983} C_VEL
LIN {X 0,Y 164.697,Z 267.508,A -85,B 0,C 180,E1 -23425.006,E2 -23425.006} C_VEL
LIN {X 0,Y 165.943,Z 270.649,A -85,B 0,C 180,E1 -23426.266,E2 -23426.266} C_VEL
LIN {X 0,Y 168.338,Z 273.427,A -85,B 0,C 180,E1 -23428.183,E2 -23428.183} C_VEL
LIN {X 0,Y 169.24,Z 274.331,A -85,B 0,C 180,E1 -23428.865,E2 -23428.865} C_VEL
LIN {X 0,Y 171.002,Z 277.914,A -85,B 0,C 180,E1 -23430.368,E2 -23430.368} C_VEL
LIN {X 0,Y 172.988,Z 280.36,A -85,B 0,C 180,E1 -23431.786,E2 -23431.786} C_VEL
LIN {X 0,Y 175.137,Z 284.351,A -85,B 0,C 180,E1 -23433.462,E2 -23433.462} C_VEL
LIN {X 0,Y 176.231,Z 285.984,A -85,B 0,C 180,E1 -23434.218,E2 -23434.218} C_VEL
LIN {X 0,Y 178.312,Z 290.002,A -85,B 0,C 180,E1 -23435.806,E2 -23435.806} C_VEL
LIN {X 0,Y 182.207,Z 298.419,A -85,B 0,C 180,E1 -23438.814,E2 -23438.814} C_VEL
LIN {X 0,Y 184.788,Z 305.157,A -85,B 0,C 180,E1 -23441,E2 -23441} C_VEL
LIN {X 0,Y 186.652,Z 312.043,A -85,B 0,C 180,E1 -23442.999,E2 -23442.999} C_VEL
LIN {X 0,Y 188.024,Z 321.989,A -85,B 0,C 180,E1 -23445.643,E2 -23445.643} C_VEL
LIN {X 0,Y 188.4,Z 331.951,A -85,B 0,C 180,E1 -23448.251,E2 -23448.251} C_VEL
LIN {X 0,Y 187.959,Z 340.396,A -85,B 0,C 180,E1 -23450.531,E2 -23450.531} C_VEL
LIN {X 0,Y 187.485,Z 345.248,A -85,B 0,C 180,E1 -23451.924,E2 -23451.924} C_VEL
LIN {X 0,Y 185.249,Z 350.892,A -85,B 0,C 180,E1 -23453.307,E2 -23453.307} C_VEL
LIN {X 0,Y 180.376,Z 361.297,A -85,B 0,C 180,E1 -23456.274,E2 -23456.274} C_VEL
LIN {X 0,Y 176.043,Z 369.885,A -85,B 0,C 180,E1 -23459.402,E2 -23459.402} C_VEL
LIN {X 0,Y 171.702,Z 378.108,A -85,B 0,C 180,E1 -23463.24,E2 -23463.24} C_VEL
LIN {X 0,Y 168.713,Z 383.803,A -85,B 0,C 180,E1 -23466.636,E2 -23466.636} C_VEL
LIN {X 0,Y 166.18,Z 388.598,A -85,B 0,C 180,E1 -23470.224,E2 -23470.224} C_VEL
LIN {X 0,Y 163.663,Z 393.494,A -85,B 0,C 180,E1 -23475.069,E2 -23475.069} C_VEL
LIN {X 0,Y 162.308,Z 396.905,A -85,B 0,C 180,E1 -23480.026,E2 -23480.026} C_VEL
LIN {X 0,Y 161.756,Z 398.923,A -85,B 0,C 180,E1 -23485.015,E2 -23485.015} C_VEL
LIN {X 0,Y 161.821,Z 399.589,A -85,B 0,C 180,E1 -23490,E2 -23490} C_VEL
LIN {X 0,Y 161.753,Z 398.902,A -85,B 0,C 180,E1 -23494.985,E2 -23494.985} C_VEL
LIN {X 0,Y 162.307,Z 396.865,A -85,B 0,C 180,E1 -23499.974,E2 -23499.974} C_VEL
LIN {X 0,Y 163.658,Z 393.433,A -85,B 0,C 180,E1 -23504.931,E2 -23504.931} C_VEL
LIN {X 0,Y 166.165,Z 388.509,A -85,B 0,C 180,E1 -23509.777,E2 -23509.777} C_VEL
LIN {X 0,Y 166.6,Z 387.692,A -85,B 0,C 180,E1 -23510.45,E2 -23510.45} C_VEL
LIN {X 0,Y 167.223,Z 385.39,A -85,B 0,C 180,E1 -23512.304,E2 -23512.304} C_VEL
LIN {X 0,Y 166.761,Z 381.281,A -85,B 0,C 180,E1 -23515.398,E2 -23515.398} C_VEL
LIN {X 0,Y 166.64,Z 376.636,A -85,B 0,C 180,E1 -23518.413,E2 -23518.413} C_VEL
LIN {X 0,Y 167.766,Z 373.489,A -85,B 0,C 180,E1 -23520.084,E2 -23520.084} C_VEL
LIN {X 0,Y 172.102,Z 365.469,A -85,B 0,C 180,E1 -23523.455,E2 -23523.455} C_VEL
LIN {X 0,Y 177.006,Z 355.993,A -85,B 0,C 180,E1 -23526.553,E2 -23526.553} C_VEL
LIN {X 0,Y 181.097,Z 347.079,A -85,B 0,C 180,E1 -23528.919,E2 -23528.919} C_VEL
LIN {X 0,Y 182.23,Z 337.49,A -85,B 0,C 180,E1 -23531.73,E2 -23531.73} C_VEL
LIN {X 0,Y 182.38,Z 326.528,A -85,B 0,C 180,E1 -23534.806,E2 -23534.806} C_VEL
LIN {X 0,Y 181.407,Z 316.371,A -85,B 0,C 180,E1 -23537.661,E2 -23537.661} C_VEL
LIN {X 0,Y 179.691,Z 309.093,A -85,B 0,C 180,E1 -23539.912,E2 -23539.912} C_VEL
LIN {X 0,Y 176.251,Z 299.604,A -85,B 0,C 180,E1 -23543.264,E2 -23543.264} C_VEL
LIN {X 0,Y 171.97,Z 290.489,A -85,B 0,C 180,E1 -23546.953,E2 -23546.953} C_VEL
LIN {X 0,Y 169.772,Z 286.463,A -85,B 0,C 180,E1 -23548.838,E2 -23548.838} C_VEL
LIN {X 0,Y 168.849,Z 284.973,A -85,B 0,C 180,E1 -23549.604,E2 -23549.604} C_VEL
LIN {X 0,Y 166.736,Z 281.502,A -85,B 0,C 180,E1 -23551.439,E2 -23551.439} C_VEL
LIN {X 0,Y 166.162,Z 280.058,A -85,B 0,C 180,E1 -23552.052,E2 -23552.052} C_VEL
LIN {X 0,Y 163.645,Z 277.12,A -85,B 0,C 180,E1 -23554.221,E2 -23554.221} C_VEL
LIN {X 0,Y 162.161,Z 273.824,A -85,B 0,C 180,E1 -23555.856,E2 -23555.856} C_VEL
LIN {X 0,Y 159.259,Z 271.095,A -85,B 0,C 180,E1 -23558.735,E2 -23558.735} C_VEL
LIN {X 0,Y 157.619,Z 267.709,A -85,B 0,C 180,E1 -23560.843,E2 -23560.843} C_VEL
LIN {X 0,Y 157.479,Z 267.126,A -85,B 0,C 180,E1 -23561.112,E2 -23561.112} C_VEL
LIN {X 0,Y 157.424,Z 266.498,A -85,B 0,C 180,E1 -23564.463,E2 -23564.463} C_VEL
LIN {X 0,Y 157.688,Z 266.458,A -85,B 0,C 180,E1 -23569.731,E2 -23569.731} C_VEL
LIN {X 0,Y 157.763,Z 266.457,A -85,B 0,C 180,E1 -23572.32,E2 -23572.32} C_VEL
LIN {X 0,Y 158.254,Z 266.396,A -85,B 0,C 180,E1 -23580,E2 -23580} C_VEL
LIN {X 0,Y 157.768,Z 266.458,A -85,B 0,C 180,E1 -23587.68,E2 -23587.68} C_VEL
LIN {X 0,Y 157.638,Z 266.472,A -85,B 0,C 180,E1 -23591.238,E2 -23591.238} C_VEL
LIN {X 0,Y 157.455,Z 266.496,A -85,B 0,C 180,E1 -23595.534,E2 -23595.534} C_VEL
LIN {X 0,Y 157.448,Z 266.684,A -85,B 0,C 180,E1 -23599.175,E2 -23599.175} C_VEL
LIN {X 0,Y 158.328,Z 269.217,A -85,B 0,C 180,E1 -23600.469,E2 -23600.469} C_VEL
LIN {X 0,Y 160.055,Z 271.269,A -85,B 0,C 180,E1 -23602.425,E2 -23602.425} C_VEL
LIN {X 0,Y 162.023,Z 272.415,A -85,B 0,C 180,E1 -23604.266,E2 -23604.266} C_VEL
LIN {X 0,Y 163.375,Z 275.328,A -85,B 0,C 180,E1 -23605.769,E2 -23605.769} C_VEL
LIN {X 0,Y 165.741,Z 277.593,A -85,B 0,C 180,E1 -23607.804,E2 -23607.804} C_VEL
LIN {X 0,Y 168.421,Z 281.928,A -85,B 0,C 180,E1 -23610.222,E2 -23610.222} C_VEL
LIN {X 0,Y 169.55,Z 283.337,A -85,B 0,C 180,E1 -23611.121,E2 -23611.121} C_VEL
LIN {X 0,Y 172.23,Z 288.071,A -85,B 0,C 180,E1 -23613.428,E2 -23613.428} C_VEL
LIN {X 0,Y 176.105,Z 295.868,A -85,B 0,C 180,E1 -23616.772,E2 -23616.772} C_VEL
